(* CODESYS project SMB_Client_Visu.project

Project tree, tasks and I/O mapping:
  Device : CODESYS Control for Raspberry Pi, 3S - Smart Software Solutions GmbH, version 3.5.12.0
    application Application
      libraries: Standard, * (System); Standard64, * (System); BASIC, 3.3.3.0 (OSCAT); File Access, 3.5.7.0 (3S - Smart Software Solutions GmbH); VisuDialogs, * (System); Network, 3.5.7.0 (3S - Smart Software Solutions GmbH); Memory, 3.5.7.0 (3S - Smart Software Solutions GmbH)
      task MainTask (cyclic, interval 4 ms, priority 1) calls PLC_PRG
      task VISU_TASK (cyclic, interval 100 ms, priority 31) calls VisuElems.Visu_Prg
      visualisation Start
      visualisation SMB_Explorer
      Bausteine/
        program PLC_PRG [CFC]
        SMB2_Client/
          Explorer/
            data type Explorer
            data type Explorer_Dummy
          Misc/
            function block DER_Encoding [ST]
            function block DER_Len [ST]
            function WSTRING_UPPER [ST]
          NTLM/
            Struct/
              data type AUTHENTICATE_MESSAGE
              data type AVPairList
              data type CHALLENGE_MESSAGE
              data type NEGOTIATE_MESSAGE
              data type SessionData
            Functions/
              Hash/Encryption/
                function block HMAC_MD5 [ST]
                function block MD4 [ST]: ROUND1, ROUND2, ROUND3
                function block RC4 [ST]
              function block ComputeResponse [ST]
              function EncryptedSessionKey [ST]
              function block GenerateAuthenticateMessage [ST]
              function GetAVPairList [ST]
              function block LMOWFv2 [ST]
              function block mechListMIC [ST]
              function block MIC [ST]
              function block NTLM [ST]
              function block NTOWFv2 [ST]
              function block ProcessChallengeMessage [ST]
              function block SEALKEY [ST]
              function SetAVPairList [ST]
              function block SIGNKEY [ST]
          SMB2/
            Functions/
              function block ReadFile [ST]
              function block SendFile [ST]
              function NetShareEnumAll [ST]
              function NetShareBind [ST]
              function decodeSharePath [ST]
              Requests/
                function CloseReq [ST]
                function CreateReq [ST]
                function LogOffReq [ST]
                function QueryDirReq [ST]
                function TreeConnectReq [ST]
                function TreeDisconnectReq [ST]
                function ReadRequest [ST]
                function NegotiateReq [ST]
            Struct/
              data type Connection
              data type Open
              data type Session
              data type SMB_Client_Error
              SMB2_Requests/
                data type SMB_COM_NEGOTIATE
                data type SMB_Dialect
                data type SMB2_CLOSE_Request
                data type SMB2_CREATE_Request
                data type SMB2_LOGOFF_Request
                data type SMB2_QUERY_DIRECTORY_Request
                data type SMB2_READ_Request
                data type SMB2_SESSION_SETUP_Request
                data type SMB2_TREE_CONNECT_Request
                data type SMB2_TREE_DISCONNECT_Request
                data type SMB2_WRITE_Request
                data type SMB2_IOCTL_Request
              SMB2_Responses/
                data type SMB2_CLOSE_Response
                data type SMB2_CREATE_Reponse
                data type SMB2_LOGOFF_Response
                data type SMB2_NEGOTIATE_Response
                data type SMB2_READ_Response
                data type SMB2_SESSION_SETUP_Response
                data type SMB2_TREE_CONNECT_Response
                data type SMB2_TREE_DISCONNECT_Response
                data type SMB2_WRITE_Response
                data type SMB2_QUERY_DIRECTORY_Response
              data type TreeConnect
              data type SMB2_FileDirectoryInfo
              data type sharePath
              Header/
                data type SMB_Header
                data type SMB2_Header_Sync
                data type SMB2_Transport_Header
          global variables Constants
          function block SMB2_Client [ST]
          global variables VAR_Explorer
    SoftMotion General Axis Pool
    I²C
    SPI
    GPIOs_A_B : GPIOs A/B, 3S - Smart Software Solutions GmbH, version 3.5.11.0
        unmapped channels: digital inputs (GPIO0..GPIO31), digital outputs (GPIO0..GPIO31)
    Onewire
    Camera device
      <Leer>
  text list GlobalTextList
*)

// Device/Application/Bausteine/SMB2_Client/Explorer/Explorer
TYPE Explorer :
STRUCT
	xExecute:BOOL:=FALSE;
	IPAdress:STRING(80):='192.168.100.150';
	User:WSTRING(80):="UserName"; // UserName Default for Guest
	Password:WSTRING(80):=""; // Password Default for Guest
	UserDomain:WSTRING(80):="CoDeSys"; // Default 
	Login:BOOL; // WebVisu Button Login
	Logout:BOOL; // WebVisu Button Logout
	open:BOOL; // WebVisu Button open
	apply:BOOL; //Button übernehmen
	folderUp:BOOL; // WebVisu Button Folder Up
	openIndex:INT; // WebVisu Index of Directory
	applyIndex:INT;	// WebVisu Index for Apply Button
	write_read:INT:=1; // Write Read Direction
	write:BOOL:=TRUE; // WebVisu Indicator for Direction
	read:BOOL:=FALSE; // WebVisu Indicator for Direction
	sharePathDecoded:sharePath;
	DirectoryIndex:INT;
	folderDepth:INT; // Depth of shared Folder - 0 = NetshareNames, >0 = Directory Names
	online:BOOL:=TRUE; // WebVisu Online Indicator
	error:BOOL:=TRUE; // WebVisu Error Indicator
	busy:BOOL; // WebVisu Busy Indicator
	done:BOOL; // WebVisu Done Indicator
	start:bool; // WebVisu Start Transfer
	Directory:ARRAY[0..127] OF WSTRING(128); // List of Shares, Directory and Files
	xdir:ARRAY[0..127] OF BOOL; // Indicates Director (0 = Dir, 1= no dir)
	xfile:ARRAY[0..127] OF BOOL; // Indicates File (0 = File, 1= no File)
	actualsharePath:WSTRING(512); // 
	copysharePath:WSTRING(512); // Sharepath on PC for automatic mode
	plcPath:STRING(512):='/var/opt/codesys/datei.xyz'; // Path on PLC SD-Card
END_STRUCT
END_TYPE

// Device/Application/Bausteine/SMB2_Client/Explorer/Explorer_Dummy
// Dummy Struct for SMB2 Client without Explorer Mode all Arrays are short for memory saving

TYPE Explorer_Dummy :
STRUCT
	xExecute:BOOL:=FALSE;
	IPAdress:STRING(80):='192.168.100.150';
	User:WSTRING(80):="UserName"; // UserName Default for Guest
	Password:WSTRING(80):=""; // Password Default for Guest
	UserDomain:WSTRING(80):="CoDeSys"; // Default 
	Login:BOOL; // WebVisu Button Login
	Logout:BOOL; // WebVisu Button Logout
	open:BOOL; // WebVisu Button open
	apply:BOOL; //Button übernehmen
	folderUp:BOOL; // WebVisu Button Folder Up
	openIndex:INT; // WebVisu Index of Directory
	applyIndex:INT;	// WebVisu Index for Apply Button
	write_read:INT:=1; // Write Read Direction
	write:BOOL:=TRUE; // WebVisu Indicator for Direction
	read:BOOL:=FALSE; // WebVisu Indicator for Direction
	sharePathDecoded:sharePath;
	DirectoryIndex:INT;
	folderDepth:INT; // Depth of shared Folder - 0 = NetshareNames, >0 = Directory Names
	online:BOOL:=TRUE; // WebVisu Online Indicator
	error:BOOL:=TRUE; // WebVisu Error Indicator
	busy:BOOL; // WebVisu Busy Indicator
	done:BOOL; // WebVisu Done Indicator
	start:bool; // WebVisu Start Transfer
	Directory:ARRAY[0..1] OF WSTRING(1); // List of Shares, Directory and Files
	xdir:ARRAY[0..1] OF BOOL; // Indicates Director (0 = Dir, 1= no dir)
	xfile:ARRAY[0..1] OF BOOL; // Indicates File (0 = File, 1= no File)
	actualsharePath:WSTRING(1); // 
	copysharePath:WSTRING(1); // Sharepath on PC for automatic mode
	plcPath:STRING(1); // Path on PLC SD-Card

END_STRUCT
END_TYPE

// Device/Application/Bausteine/SMB2_Client/NTLM/Struct/AUTHENTICATE_MESSAGE
{attribute 'pack_mode' := '1'} (*aligned to byte*)

TYPE AUTHENTICATE_MESSAGE :
STRUCT
	Signature:STRING(7):='NTLMSSP';
	MessageType:DWORD:=16#0003;
	// LmChallengeResponse
	LmChallengeResponseLen:WORD;
	LmChallengeResponseMaxLen:WORD;
	LmChallengeResponseBufferOffset:DWORD;
	// NtChallengeResponse
	NtChallengeResponseLen:WORD;
	NtChallengeResponseMaxLen:WORD;
	NtChallengeResponseBufferOffset:DWORD;
	// Domain Name
	DomainNameLen:WORD;
	DomainNameMaxLen:WORD;
	DomainNameBufferOffset:DWORD;
	// User Name
	UserNameLen:WORD;
	UserNameMaxLen:WORD;
	UserNameBufferOffset:DWORD;
	// Workstation
	WorkstationLen:WORD;
	WorkstationMaxLen:WORD;
	WorkstationBufferOffset:DWORD;
	// EncryptedRandomSessionKey
	EncryptedRandomSessionKeyLen:WORD;
	EncryptedRandomSessionKeyMaxLen:WORD;
	EncryptedRandomSessionKeyBufferOffset:DWORD;
	//
	NegotiateFlags:DWORD; // Negotiate Flags
	Version:ARRAY[0..1] OF DWORD:=[16#3839000A, 16#F0000000]; // Verson Number
	MIC:ARRAY[0..15] OF BYTE; // Message Integrity Code
	Payload:ARRAY[0..1023] OF BYTE; // Payload for Names and Attributes
	PayLoadSize:INT; // Length of Payload
END_STRUCT
END_TYPE

// Device/Application/Bausteine/SMB2_Client/NTLM/Struct/AVPairList
TYPE AVPairList :
STRUCT
	NBComputerName:WSTRING(80); // 
	NBDomainName:WSTRING(80);
	DNSComputerName:WSTRING(80);
	DNSDomainName:WSTRING(80);
	xTimeStamp:BOOL; // Timestamp is there
	TimeStamp:ARRAY[0..7] OF BYTE;
END_STRUCT
END_TYPE

// Device/Application/Bausteine/SMB2_Client/NTLM/Struct/CHALLENGE_MESSAGE
{attribute 'pack_mode' := '1'} (*aligned to byte*)

TYPE CHALLENGE_MESSAGE :
STRUCT
	Signature:STRING(7); // NTLMSSP
	MessageType:DWORD; // Challenge MEssage
	// TargetNameFields
	TargetNameLen:WORD;
	TargetNameMaxLen:WORD;
	TargetNameBufferOffset:DWORD;
	//
	NegotiateFlags:DWORD; // NEgotiate Flags
	ServerChallenge:ARRAY[0..7] OF BYTE; // Random Numbers Server Challenge
	Reserved:ARRAY[0..7] OF BYTE;
	// TargetInfoFields
	TargetInfoLen:WORD;
	TargetInfoMaxLen:WORD;
	TargetInfoBufferOffset:DWORD;
	//
	Version:ARRAY[0..1] OF DWORD; // Version Number
	// Payload
	TargetName:WSTRING(80);
	AVPairList:AVPairList;
	AVPairListPayload:ARRAY[0..255] OF BYTE;
END_STRUCT
END_TYPE

// Device/Application/Bausteine/SMB2_Client/NTLM/Struct/NEGOTIATE_MESSAGE
{attribute 'pack_mode' := '1'} (*aligned to byte*)

TYPE NEGOTIATE_MESSAGE :
STRUCT
	Signature:STRING(7):= 'NTLMSSP'; // NTLMSSP
	MessageType:DWORD:=16#00000001; // Negotiate MEssage
	NegotiateFlags:DWORD; // Negotiate Flags
	// Doman Name
	DomainNameLen:WORD; 
	DomainNameMaxLen:WORD;
	DomainNameBufferOffset:DWORD;
	// Workstation Name
	WorkstationLen:WORD;
	WorkstationMaxLen:WORD;
	WorkstationBufferOffset:DWORD;
	Version:ARRAY[0..1] OF DWORD:=[16#3839000a, 16#F0000000] ; // Version
END_STRUCT
END_TYPE

// Device/Application/Bausteine/SMB2_Client/NTLM/Struct/SessionData
TYPE SessionData :
STRUCT
//	mode Mode

	user:WSTRING(80); // Username
	password:WSTRING(80); // Password
	userDomain:WSTRING(80); // User Doman

	NegotiateFlags:DWORD; // Negotiate Flags

	negotiateMessage:POINTER TO NEGOTIATE_MESSAGE; // Pointer to Negotiate Message
	challengeMessage:POINTER TO CHALLENGE_MESSAGE; // Pointer to Challenge Message
//	authenticateMessage *AuthenticateMessage

	serverChallenge:ARRAY[0..7] OF BYTE; // Server Challenge random number
	clientChallenge:ARRAY[0..7] OF BYTE; // client Challenge for response
	ntChallengeResponse:ARRAY[0..511] OF BYTE; // NT Challenge Response
	ntChallengeResponseLen:WORD;  // Length of NT Challenge Response
	lmChallengeResponse:ARRAY[0..511] OF BYTE;  // LM Challenge Response
	lmChallengeResponseLen:WORD; // Length of LM Challenge Response

	responseKeyLM: ARRAY[0..15] OF BYTE; // Response Key LM for calculation
	responseKeyNT: ARRAY[0..15] OF BYTE; // Response Key NT for calculation
	exportedSessionKey: ARRAY[0..15] OF BYTE; // exported Session Key
	encryptedRandomSessionKey: ARRAY[0..15] OF BYTE; // encrypted Random Session Key
	keyExchangeKey:ARRAY[0..15] OF BYTE; // Key Exchange Key
	sessionBaseKey:ARRAY[0..15] OF BYTE; // Session Base Key
	mic                 :ARRAY[0..15] OF BYTE; // Message Integrity Code

	ClientSigningKey: ARRAY[0..15] OF BYTE; // Client Signing Key
	ServerSigningKey: ARRAY[0..15] OF BYTE; // Server Signing Key
	ClientSealingKey: ARRAY[0..15] OF BYTE; // Client Sealing Key
	ServerSealingKey: ARRAY[0..15] OF BYTE; // Server Sealing Key

	clientHandle:RC4;
	serverHandle:RC4;
	
	NegMessByte:ARRAY[0..511] OF BYTE;
	NegMessByteLen:INT;
	ChallMessByte:ARRAY[0..511] OF BYTE;
	ChallMessByteLen:INT;
	AuthMessByte:ARRAY[0..511] OF BYTE;
	AuthMessByteLen:INT;
	
	mechListMIC:ARRAY[0..19] OF BYTE;
END_STRUCT
END_TYPE

// Device/Application/Bausteine/SMB2_Client/SMB2/Struct/Connection
TYPE Connection :
STRUCT
	Session:Session; // Parameter of active Session
	MaxTransactSize:DWORD; // Max Transaction Size
	MaxReadSize:DWORD; // Max Read Size from Server
	MaxWriteSize:DWORD;	// Max Write Size to Server
	MessageID: ARRAY[0..1] OF DWORD; // Sequence Number
	ServerGuid:ARRAY [0..3] OF DWORD; // Server global unique identifier
	RequireSigning:BOOL;
	LastStatus:DWORD; // Last Status of Response
	ServerName:STRING(80); // Servername
	wServerName:WSTRING(80); // Servername Unicode String
	User:WSTRING(80); // Username
	Password:WSTRING(80); // Password
	UserDomain:WSTRING(80); // User Domain
	requestedFileName:WSTRING(512); // requested File Name
END_STRUCT
END_TYPE

// Device/Application/Bausteine/SMB2_Client/SMB2/Struct/Open
TYPE Open :
STRUCT
	FileId:ARRAY[0..3] OF DWORD; // File ID of opened File (After Create Request)
	FileSize:ARRAY[0..1] OF DWORD; // File Size of opened File (After Create Request)
	ReadDataOffset:BYTE; // Actual Offset in opened File
	ReadDataLength:DWORD; // Actual Size of read Data
END_STRUCT
END_TYPE

// Device/Application/Bausteine/SMB2_Client/SMB2/Struct/Session
TYPE Session :
STRUCT
	SessionID:ARRAY[0..1] OF DWORD; // Session ID of active Session
	TreeConnect: TreeConnect; // Parameter of Active Tree
	SessionKey:ARRAY[0..15] OF BYTE; 
	SigningRequired:BOOL;
	Open:Open;
END_STRUCT
END_TYPE

// Device/Application/Bausteine/SMB2_Client/SMB2/Struct/SMB_Client_Error
TYPE SMB_Client_Error :
STRUCT
	Error_1:INT; // Error Step in SMB2 Client 
	Error_2:DWORD; // Error/Status from Response
	TCP:NBS.ERROR; // Error TCP Function
	ConRST:BOOL; // Connection Reset from Server
END_STRUCT
END_TYPE

// Device/Application/Bausteine/SMB2_Client/SMB2/Struct/SMB2_Requests/SMB_COM_NEGOTIATE
{attribute 'pack_mode' := '1'} (*aligned to byte*)

TYPE SMB_COM_NEGOTIATE :	
STRUCT
	WORDCOUNT :BYTE;
	BYTECOUNT :WORD;
	Dialects: ARRAY[0..8] OF SMB_Dialect;
END_STRUCT
END_TYPE

// Device/Application/Bausteine/SMB2_Client/SMB2/Struct/SMB2_Requests/SMB_Dialect
{attribute 'pack_mode' := '1'} (*aligned to byte*)

TYPE SMB_Dialect :
STRUCT
	BufferFormat:BYTE;
	DialectString:STRING;
END_STRUCT
END_TYPE

// Device/Application/Bausteine/SMB2_Client/SMB2/Struct/Header/SMB_Header
{attribute 'pack_mode' := '1'} (*aligned to byte*)

TYPE SMB_Header :
STRUCT
	Protocol: ARRAY[0..3] OF BYTE;
	Command: BYTE;
	Status:DWORD;
	Flags:BYTE;
	Flags2:WORD;
	PIDHigh:WORD;
	SecurityFeatures:ARRAY[0..7] OF BYTE;
	Reserved:WORD;
	TID:WORD;
	PIDLow:WORD;
	UID:WORD;
	MID:WORD;
END_STRUCT
END_TYPE

// Device/Application/Bausteine/SMB2_Client/SMB2/Struct/Header/SMB2_Header_Sync
// [MS-SMB2] 2.2.1.2
{attribute 'pack_mode' := '1'} (*aligned to byte*)

TYPE SMB2_Header_Sync :
STRUCT
	ProtocolID: ARRAY[0..3] OF BYTE;
	StructureSize:WORD:=64;
	CreditCharge:WORD;
	Status:DWORD;
	Command:WORD;
	CreditRepReq:WORD;
	Flags: DWORD;
	NextCommand:DWORD;
	MessageID: ARRAY[0..1] OF DWORD;
	Reserved: DWORD;
	TreeID:DWORD;
	SessionID: ARRAY[0..1] OF DWORD;
	Signature: ARRAY[0..3] OF DWORD;
END_STRUCT
END_TYPE

// Device/Application/Bausteine/SMB2_Client/SMB2/Struct/SMB2_Requests/SMB2_CLOSE_Request
// [MS-SMB2] 2.2.15

{attribute 'pack_mode' := '1'} (*aligned to byte*)

TYPE SMB2_CLOSE_Request :
STRUCT
	StructureSize:WORD:=24;
	Flags:WORD;
	Reserved:DWORD:=0;
	FileId:ARRAY[0..3] OF DWORD;
END_STRUCT
END_TYPE

// Device/Application/Bausteine/SMB2_Client/SMB2/Struct/SMB2_Requests/SMB2_CREATE_Request
// [MS-SMB2] 2.2.13

{attribute 'pack_mode' := '1'} (*aligned to byte*)

TYPE SMB2_CREATE_Request :
STRUCT
	StructureSize:WORD:=57;
	SecurityFlags:BYTE;
	RequestedOplockLevel:BYTE;
	ImpersonationLevel:DWORD;
	SmbCreateFlags:ARRAY[0..1] OF DWORD;
	Reserved:ARRAY[0..1] OF DWORD;
	DesiredAccess:DWORD;
	FileAttributes:DWORD;
	ShareAccess:DWORD;
	CreateDisposition:DWORD;
	CreateOptions:DWORD;
	NameOffset:WORD;
	NameLength:WORD;
	CreateContextsOffset:DWORD;
	CreateContextsLength:DWORD;
	Payload:ARRAY[0..255] OF BYTE;
END_STRUCT
END_TYPE

// Device/Application/Bausteine/SMB2_Client/SMB2/Struct/SMB2_Requests/SMB2_LOGOFF_Request
// [MS-SMB2] 2.2.7

{attribute 'pack_mode' := '1'} (*aligned to byte*)

TYPE SMB2_LOGOFF_Request :
STRUCT
	StructureSize:WORD;
	Reserved:WORD;
END_STRUCT
END_TYPE

// Device/Application/Bausteine/SMB2_Client/SMB2/Struct/SMB2_Requests/SMB2_QUERY_DIRECTORY_Request
// [MS-SMB2] 2.2.33

{attribute 'pack_mode' := '1'} (*aligned to byte*)

TYPE SMB2_QUERY_DIRECTORY_Request :
STRUCT
	StructureSize:WORD:=33;
	FileInformationClass:BYTE;
	Flags:BYTE;
	FileIndex:DWORD;
	FileId:ARRAY[0..3] OF DWORD;
	FileNameOffset:WORD;
	FileNameLength:WORD;
	OutputbufferLength:DWORD;
	Payload:ARRAY[0..127] OF BYTE;
END_STRUCT
END_TYPE

// Device/Application/Bausteine/SMB2_Client/SMB2/Struct/SMB2_Requests/SMB2_READ_Request
// [MS-SMB2] 2.2.19

{attribute 'pack_mode' := '1'} (*aligned to byte*)

TYPE SMB2_READ_Request :
STRUCT
	StructureSize:WORD:=49;
	Padding:BYTE; // Offset in Response from Header Start ( for data optimization)
	Flags:BYTE:=0; // Not used in SMB 2
	Length:DWORD; // Length of data to read
	Offset:LWORD; // Offset in File
	FileId:ARRAY[0..3] OF DWORD;
	MinimumCount:DWORD; // Minimal number of Bytes to be read for success
	Channel:DWORD:=0; // SMB2 = 0;
	RemainingBytes:DWORD; // Number of Bytes to be read after this operation completes
	ReadChannelInfoOffset:WORD:=0; // SMB2 = 0;
	ReadChannelInfoLength:WORD:=0; // SMB2 = 0;
END_STRUCT
END_TYPE

// Device/Application/Bausteine/SMB2_Client/SMB2/Struct/SMB2_Requests/SMB2_SESSION_SETUP_Request
// [MS-SMB2] 2.2.5

{attribute 'pack_mode' := '1'} (*aligned to byte*)

TYPE SMB2_SESSION_SETUP_Request :
STRUCT
	StructureSize:WORD;
	Flags:BYTE;
	SecurityMode:BYTE;
	Capabilities:DWORD;
	Channel:DWORD;
	SecurityBufferOffset:WORD;
	SecurityBufferLength:WORD;
	PrevSessionsId:ARRAY[0..1] OF DWORD;
END_STRUCT
END_TYPE

// Device/Application/Bausteine/SMB2_Client/SMB2/Struct/SMB2_Requests/SMB2_TREE_CONNECT_Request
// [MS-SMB2] 2.2.9

{attribute 'pack_mode' := '1'} (*aligned to byte*)

TYPE SMB2_TREE_CONNECT_Request :
STRUCT
	StructureSize:WORD;
	Flags:WORD;
	PathOffset:WORD;
	PathLength:WORD;
	PathName:WSTRING(256);
END_STRUCT
END_TYPE

// Device/Application/Bausteine/SMB2_Client/SMB2/Struct/SMB2_Requests/SMB2_TREE_DISCONNECT_Request
// [MS-SMB2] 2.2.11

{attribute 'pack_mode' := '1'} (*aligned to byte*)

TYPE SMB2_TREE_DISCONNECT_Request :
STRUCT
	StructureSize:WORD;
	Reserved:WORD;
END_STRUCT
END_TYPE

// Device/Application/Bausteine/SMB2_Client/SMB2/Struct/SMB2_Requests/SMB2_WRITE_Request
// [MS-SMB2] 2.2.21

{attribute 'pack_mode' := '1'} (*aligned to byte*)

TYPE SMB2_WRITE_Request :
STRUCT
	StructureSize:WORD:=49;
	DataOffset:WORD;
	Length:DWORD;
	Offset:LWORD;
	FileId:ARRAY[0..3] OF DWORD;
	Channel:DWORD:=0; // SMB2 = 0;
	RemainingBytes:DWORD;
	WriteChannelInfoOffset:WORD:=0; // SMB2 = 0;
	WriteChannelInfoLength:WORD:=0; // SMB2 = 0;
	Flags:DWORD:=0; // SMB2 = 0;
END_STRUCT
END_TYPE

// Device/Application/Bausteine/SMB2_Client/SMB2/Struct/SMB2_Responses/SMB2_CLOSE_Response
// [MS-SMB2] 2.2.16

{attribute 'pack_mode' := '1'} (*aligned to byte*)

TYPE SMB2_CLOSE_Response :
STRUCT
	StructureSize:WORD;
	Flags:WORD;
	Reserved:DWORD;
	CreateionTime:ARRAY[0..1] OF DWORD;
	LastAccessTime:ARRAY[0..1] OF DWORD;
	LastWriteTime:ARRAY[0..1] OF DWORD;
	ChangeTime:ARRAY[0..1] OF DWORD;
	AllocationSize:ARRAY[0..1] OF DWORD;
	EndofFile:ARRAY[0..1] OF DWORD;
	FileAttributes:DWORD;
END_STRUCT
END_TYPE

// Device/Application/Bausteine/SMB2_Client/SMB2/Struct/SMB2_Responses/SMB2_CREATE_Reponse
// [MS-SMB2] 2.2.114

{attribute 'pack_mode' := '1'} (*aligned to byte*)

TYPE SMB2_CREATE_Reponse :
STRUCT
	StructureSize:WORD;
	OplockLevel:BYTE;
	Flags:BYTE;
	CreateAction:DWORD;
	CreateionTime:ARRAY[0..1] OF DWORD;
	LastAccessTime:ARRAY[0..1] OF DWORD;
	LastWriteTime:ARRAY[0..1] OF DWORD;
	ChangeTime:ARRAY[0..1] OF DWORD;
	AllocationSize:ARRAY[0..1] OF DWORD;
	EndofFile:ARRAY[0..1] OF DWORD;
	FileAttributes:DWORD;
	Reserved2:DWORD;
	FileId:ARRAY[0..3] OF DWORD;
	CreateContextsOffset:DWORD;
	CreateContextsLength:DWORD;
END_STRUCT
END_TYPE

// Device/Application/Bausteine/SMB2_Client/SMB2/Struct/SMB2_Responses/SMB2_LOGOFF_Response
// [MS-SMB2] 2.2.8

{attribute 'pack_mode' := '1'} (*aligned to byte*)

TYPE SMB2_LOGOFF_Response :
STRUCT
	StructureSize:WORD;
	Reserved:WORD;
END_STRUCT
END_TYPE

// Device/Application/Bausteine/SMB2_Client/SMB2/Struct/SMB2_Responses/SMB2_NEGOTIATE_Response
// [MS-SMB2] 2.2.4

{attribute 'pack_mode' := '1'} (*aligned to byte*)

TYPE SMB2_NEGOTIATE_Response :
STRUCT
	StructureSize:WORD;
	SecurityMode:WORD;
	DialectRevision:WORD;
	NegotiateContextCount:WORD;
	ServerGuid:ARRAY [0..3] OF DWORD;
	Capabilities:DWORD;
	MaxTransactSize:DWORD;
	MaxReadSize:DWORD;
	MaxWriteSize:DWORD;
	SystemTime:ARRAY[0..1] OF DWORD;
	ServerStartTime:ARRAY[0..1] OF DWORD;
	SecurityBufferOffset:WORD;
	SecurityBufferLength:WORD;
	NegotiateContextOffset:DWORD;
	
END_STRUCT
END_TYPE

// Device/Application/Bausteine/SMB2_Client/SMB2/Struct/SMB2_Responses/SMB2_READ_Response
// [MS-SMB2] 2.2.20

{attribute 'pack_mode' := '1'} (*aligned to byte*)

TYPE SMB2_READ_Response :
STRUCT
	StructureSize:WORD;
	DataOffset:BYTE; // Data Offset in Response Buffer from SMB2 Header
	Reserved:BYTE;
	DataLength:DWORD;
	DataRemaining:DWORD;
	Reserved2:DWORD;
END_STRUCT
END_TYPE

// Device/Application/Bausteine/SMB2_Client/SMB2/Struct/SMB2_Responses/SMB2_SESSION_SETUP_Response
// [MS-SMB2] 2.2.6

{attribute 'pack_mode' := '1'} (*aligned to byte*)

TYPE SMB2_SESSION_SETUP_Response :
STRUCT
	StructureSize:WORD;
	SessionFlags:WORD;
	SecurityBufferOffset:WORD;
	SecurityBufferLength:WORD;
END_STRUCT
END_TYPE

// Device/Application/Bausteine/SMB2_Client/SMB2/Struct/SMB2_Responses/SMB2_TREE_CONNECT_Response
// [MS-SMB2] 2.2.10

{attribute 'pack_mode' := '1'} (*aligned to byte*)

TYPE SMB2_TREE_CONNECT_Response :
STRUCT
	StructureSize:WORD;
	ShareType:BYTE;
	Reserved:BYTE;
	ShareFlags:DWORD;
	Capabilities:DWORD;
	MaxmalAccess:DWORD;
END_STRUCT
END_TYPE

// Device/Application/Bausteine/SMB2_Client/SMB2/Struct/SMB2_Responses/SMB2_TREE_DISCONNECT_Response
// [MS-SMB2] 2.2.12

{attribute 'pack_mode' := '1'} (*aligned to byte*)

TYPE SMB2_TREE_DISCONNECT_Response :
STRUCT
	StructureSize:WORD;
	Reserved:WORD;
END_STRUCT
END_TYPE

// Device/Application/Bausteine/SMB2_Client/SMB2/Struct/SMB2_Responses/SMB2_WRITE_Response
// [MS-SMB2] 2.2.22

{attribute 'pack_mode' := '1'} (*aligned to byte*)

TYPE SMB2_WRITE_Response :
STRUCT
	StructureSize:WORD;
	Reserved:WORD; 
	Count:DWORD; // Number of written Bytes
	Remaining:DWORD; // Must be 0
	WriteChannelInfoOffset:WORD; // Must be 0
	WriteChannelInfoLength:WORD; // Must be 0
END_STRUCT
END_TYPE

// Device/Application/Bausteine/SMB2_Client/SMB2/Struct/Header/SMB2_Transport_Header
// [MS-SMB2] 2.1

{attribute 'pack_mode' := '1'} (*aligned to byte*)

TYPE SMB2_Transport_Header :
STRUCT
	Zero:BYTE; (*Always Zero, for Direct TCP Transport*)
	StreamProtocolLength:UDINT; (*Length of SMB2 Packet without Transport Header*)
END_STRUCT
END_TYPE

// Device/Application/Bausteine/SMB2_Client/SMB2/Struct/TreeConnect
TYPE TreeConnect :
STRUCT
	ShareName:WSTRING(128); // Name of Share Name
	TreeConnectId:DWORD; // TreeID of opened Tree
	IsDfsShare:BOOL;
END_STRUCT
END_TYPE

// Device/Application/Bausteine/SMB2_Client/SMB2/Struct/SMB2_FileDirectoryInfo
{attribute 'pack_mode' := '1'} (*aligned to byte*)

TYPE SMB2_FileDirectoryInfo :
STRUCT
	NextOffset:DWORD; // Offset to Next File Directory Info
	FileIndex:DWORD; // File Index Number
	Create:LWORD; // Create Time
	LastAcc:LWORD; // Last Access Time
	LastWrite:LWORD; // Last Write Time
	LastChange:LWORD; // Last Change Time
	EndOfFile:LWORD; // End of File in Byte
	AllocSize:LWORD; // Allocation Size on Disk
	FileAtr:DWORD; // File Attributes
	FileNameLength:DWORD; // Length of File Name
END_STRUCT
END_TYPE

// Device/Application/Bausteine/SMB2_Client/SMB2/Struct/SMB2_Responses/SMB2_QUERY_DIRECTORY_Response
// [MS-SMB2] 2.2.34

{attribute 'pack_mode' := '1'} (*aligned to byte*)

TYPE SMB2_QUERY_DIRECTORY_Response :
STRUCT
	StructureSize:WORD;
	OutputBufferOffset:WORD;
	OutputBufferLength:DWORD;
END_STRUCT
END_TYPE

// Device/Application/Bausteine/SMB2_Client/SMB2/Struct/SMB2_Requests/SMB2_IOCTL_Request
// [MS-SMB2] 2.2.31

{attribute 'pack_mode' := '1'} (*aligned to byte*)

TYPE SMB2_IOCTL_Request :
STRUCT
	StructureSize:WORD;
	Reserved:WORD;
	CtlCode:DWORD;
	FileID:ARRAY[0..3] OF DWORD;
	InputOffset:DWORD;
	InputCount:DWORD;
	MaxInputResponse:DWORD;
	OutputOffset:DWORD;
	OutputCount:DWORD;
	MaxOutputResponse:DWORD;
	Flags:DWORD;
	Reserved2:DWORD;
END_STRUCT
END_TYPE

// Device/Application/Bausteine/SMB2_Client/SMB2/Struct/sharePath
TYPE sharePath :
STRUCT
	serverName:WSTRING(64); // ServerName or IP Adress - max 64 Symbols
	treeName:WSTRING(256); // ShareName of shared Folder - max 256 Symbols
	fileName:WSTRING(512); // Filename - \folder\folder_2\filename.x
END_STRUCT
END_TYPE

// Device/Application/Bausteine/SMB2_Client/Constants
{attribute 'qualified_only'}
VAR_GLOBAL CONSTANT
	(*SMB2 Header Commands*)
	NEGOTIATE 			:UINT:= 16#0000;
	SESSION_SETUP 		:UINT:= 16#0001;
	LOGOFF 				:UINT:= 16#0002;
	TREE_CONNECT 		:UINT:= 16#0003;
	TREE_DISCONNECT 	:UINT:= 16#0004;
	CREATE 				:UINT:= 16#0005;
	CLOSE 				:UINT:= 16#0006;
	FLUSH 				:UINT:= 16#0007;
	READ 				:UINT:= 16#0008;
	WRITE 				:UINT:= 16#0009;
	LOCK 				:UINT:= 16#000A;
	IOCTL 				:UINT:= 16#000B;
	CANCEL 				:UINT:= 16#000C;
	ECHO 				:UINT:= 16#000D;
	QUERY_DIRECTORY 	:UINT:= 16#000E;
	CHANGE_NOTIFY 		:UINT:= 16#000F;
	QUERY_INFO 			:UINT:= 16#0010;
	SET_INFO 			:UINT:= 16#0011;
	OPLOCK_BREAK 		:UINT:= 16#0012;
	(*SMB2 Header Flags*)
	SMB2_FLAGS_SERVER_TO_REDIR 			:UDINT:= 16#00000001;
	SMB2_FLAGS_ASYNC_COMMAND 			:UDINT:= 16#00000002;
	SMB2_FLAGS_RELATED_OPERATIONS 		:UDINT:= 16#00000004;
	SMB2_FLAGS_SIGNED 					:UDINT:= 16#00000008;
	SMB2_FLAGS_PRIORITY_MASK 			:UDINT:= 16#00000070;
	SMB2_FLAGS_DFS_OPERATIONS 			:UDINT:= 16#10000000;
	SMB2_FLAGS_REPLAY_OPERATION 		:UDINT:= 16#20000000;
	
	(*SMB Flags*)
	SMB_FLAGS_LOCK_AND_READ_OK 			:USINT:= 16#01;
	SMB_FLAGS_BUF_AVAIL 				:USINT:= 16#02;
	SMB_FLAGS_CASE_INSENSITIVE 			:USINT:= 16#08;
	SMB_FLAGS_CANONICALIZED_PATHS 		:USINT:= 16#10;
	SMB_FLAGS_OPLOCK 					:USINT:= 16#20;
	SMB_FLAGS_OPBATCH 					:USINT:= 16#40;
	SMB_FLAGS_REPLY						:USINT:= 16#80;
	
	SMB_FLAGS2_LONG_NAMES				:UINT:= 16#0001;
	SMB_FLAGS2_EAS						:UINT:= 16#0002;
	SMB_FLAGS2_SMB_SECURITY_SIGNATURE 	:UINT:= 16#0004;
	SMB_FLAGS2_IS_LONG_NAME				:UINT:= 16#0040;
	SMB_FLAGS2_DFS						:UINT:= 16#1000;
	SMB_FLAGS2_PAGING_IO 				:UINT:= 16#2000;
	SMB_FLAGS2_NT_STATUS 				:UINT:= 16#4000;
	SMB_FLAGS2_UNICODE 					:UINT:= 16#8000;
	
	(*Header Status*)
	STATUS_SUCCESS						:UDINT:= 16#00000000;
	STATUS_MORE_PROCESSING_REQUIRED		:UDINT:= 16#C0000016;
END_VAR

// Device/Application/Bausteine/SMB2_Client/VAR_Explorer
{attribute 'qualified_only'}
VAR_GLOBAL RETAIN
	Visu_Explorer:explorer;
END_VAR

// Device/Application/Bausteine/PLC_PRG
PROGRAM PLC_PRG
VAR
	SMB2: SMB2_Client; // SMB2 Client
	start:BOOL; // Start for Automatic Mode (or for testing)
	done:BOOL;	// File Transfer Done or Explorer Mode LogOff Done
	busy:BOOL; // File Transfer active or Explorer Mode connected to Server
	error:BOOL; // Error
	eError:SMB_Client_Error; // Error Struct for detailed error information
END_VAR

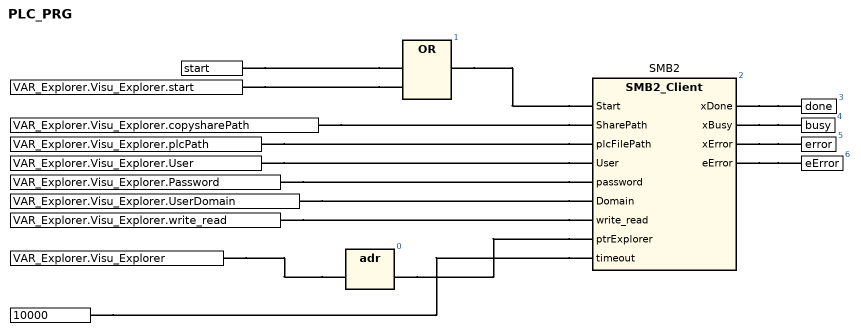
SMB2(
    Start := start OR VAR_Explorer.Visu_Explorer.start,
    SharePath := VAR_Explorer.Visu_Explorer.copysharePath,
    plcFilePath := VAR_Explorer.Visu_Explorer.plcPath,
    User := VAR_Explorer.Visu_Explorer.User,
    password := VAR_Explorer.Visu_Explorer.Password,
    Domain := VAR_Explorer.Visu_Explorer.UserDomain,
    write_read := VAR_Explorer.Visu_Explorer.write_read,
    ptrExplorer := adr(VAR_Explorer.Visu_Explorer),
    timeout := 10000); // SMB2_Client
done := SMB2.xDone;
busy := SMB2.xBusy;
error := SMB2.xError;
eError := SMB2.eError;

END_PROGRAM

// Device/Application/Bausteine/SMB2_Client/SMB2_Client
FUNCTION_BLOCK SMB2_Client
VAR_INPUT
	Start:BOOL;					// Starts Connection and Write/Read process
	SharePath:WSTRING(256);		// shared folder Path, with Ip Adress - \\IP Adress\share\subfolder\filename.x
	plcFilePath:STRING(256);	// Path and Name of File in the PLC - manufactur / OS specific
	User:WSTRING(80);			// User Name - for Guest choose any User Name
	password:WSTRING(80);		// User Password for User Name - "Password01" - for Guest use empty WSTRING ""
	Domain:WSTRING(80); 		// Domain Name of PLC, for default use "CoDeSys"
	write_read:INT; 			// 1 = write file from PLC Memory to Shared Folder , 2 = read file from Shared Folder to PLC Memory
	ptrExplorer:POINTER TO Explorer; // Pointer to Explorer Variable for WebVisu Explorer
	timeout:UINT; // Timeout in ms
END_VAR
VAR_OUTPUT
	xDone:BOOL; // send/receive done or explorer mode log off done
	xBusy:BOOL;	// send/receive busy or explorer mode active
	xError:BOOL; // error
	eError:SMB_Client_Error; // error struct for detailed error information
	
END_VAR
VAR
	ConnectionParam:Connection; // Connection Parameter
	sharePathDecoded:sharePath; // SharePath decoded in ServerName, TreeName and FileName
	explorerDummy:Explorer_Dummy; // Explorer Dummy Variable when no Explorer used
	explorerMode:BOOL; // Indicates Explorer active
	explorerVar:BOOL:=FALSE;
	
	step:INT;	// actual step
	lastStep:INT; // step last cycle - for timeout
	errorStep:INT; // step of error
	timeoutTON:TON; // timeout timer
	autoLogOffTON:TON; // Automactic LogOff in WebVisu after x Minutes
	
	lastActive:BOOL; // 
	(*Connection*)
	TCP1: NBS.TCP_Client; // TCP Client Funtcion
	hCon:CAA.handle; // Handle to TCP Connection, for read and write
	Erro: NBS.ERROR; // TCP Error
	active:BOOL; // Indicates active TCP connection
	(*Receive TCP*)
	TCPRECV: NBS.TCP_Read; // TCP Receive Function
	recvP:CAA.PVOID:=ADR(recvBuf); // Pointer to Receive Buffer
	recvBuf: ARRAY[0..BufferSize+1024] OF BYTE; // receive buffer
	recvComplete:BOOL; // Received and copied to Response Variables
	recvOK:BOOL; // All TCP Segments received, ready for copy to variables
	(*Receive fragmeted TCP Packets*)
	MessageLength:UDINT; // Message Length in Header
	recvLength:UDINT; // Received Data Length
	newBufferIndex:UDINT; // Start for next received data, used for fragmented TCP
	
	(*Write TCP*)
	TCPSEND: NBS.TCP_WRITE; // TCP Send Function
	sendBuf: ARRAY[0..BufferSize+1024] OF BYTE; // send buffer
	sendP: CAA.PVOID:=ADR(sendBuf); // Pointer to Send Buffer
	sendSize: CAA.SIZE; // Length of Send Buffer
	sendS:uint;
	startSend: BOOL; // Start Sending
	
	(*SMB Responses*)
	TransportHeader:SMB2_Transport_Header;
	TransportHeaderRep:SMB2_Transport_Header;
	SMB2Header: SMB2_Header_Sync;
	SMB2HeaderRep: SMB2_Header_Sync;
	SMBHeader: SMB_Header;
	SMBNegotiate:SMB_COM_NEGOTIATE;
	SMB2NegotiateRep:SMB2_NEGOTIATE_Response;
	SMB2SessionSetup:SMB2_SESSION_SETUP_Request;
	SMB2SessionSetupRep:SMB2_SESSION_SETUP_Response;
	SMB2TreeConnectRep:SMB2_TREE_CONNECT_Response;
	SMB2CreateRep:SMB2_CREATE_Reponse;
	SMB2ReadRep:SMB2_READ_Response;
	SMB2WriteRep:SMB2_WRITE_Response;
	SMB2CloseRep:SMB2_CLOSE_Response;
	SMB2DisconnectRep:SMB2_TREE_DISCONNECT_Response;
	SMB2LogoffRep:SMB2_LOGOFF_Response;
	SMB2QueryDirRep:SMB2_QUERY_DIRECTORY_Response;
	tmpFileDirectoryInfo:SMB2_FileDirectoryInfo;
	
	repSize:UINT; // Size of received Data - Transport Header
	repP:POINTER TO BYTE;
	tmpIndex:UINT;
	repIndex:UINT;
	startIndex:UINT;

	sendF:sendFile; // Send File to Server
	readF:ReadFile; // Receive File from Server
	NTLM:NTLM; // NTLM Function Block
	
	i:DINT;
	j:INT;
	h:INT;
	
	// explorer mode variable
	varPtr:POINTER TO ARRAY[0..9216] OF BYTE;
	stringPtr:POINTER TO ARRAY[0..1024] OF BYTE;
	tempOffset:DINT;	
	tempLen:UINT;
	numberOfNames:INT;	
	pVar:POINTER TO ARRAY[0..1024] OF BYTE;
	pWord:POINTER TO ARRAY[0..1024] OF WORD;
	pLWORD:POINTER TO ARRAY[0..7] OF BYTE;
	tempLWORD:LWORD;
	tempLWORD2:LWORD;
	tempwString:WSTRING(512);
END_VAR
VAR CONSTANT
	BufferSize:UDINT:= 16384;//8192//32768//16384 - Buffersize for send and receive Buffer
END_VAR

// This is the Main SMB2_Client Function
// Normal Mode: File Transfer in Both Direction PLC - > PC and PC -> PLC. Both diretions initiates by PLC.
// Explorer Mode in HMI for browsing trough Shared Folders and setting new Share Path for Automatic Mode.

// Timeout
timeoutTON(PT:=UINT_TO_TIME(timeout));

IF (step = laststep) AND NOT (step=01) AND NOT (step=500) THEN // Start Timer when same step
	timeoutTON.IN := TRUE;
ELSE
	timeoutTON.IN := FALSE;
END_IF
lastStep := step;

IF timeoutTON.Q THEN // Timeout -> Error
	errorStep:=step;
	step:=900;
END_IF


// Copy Dummy Explorervariable when Explorer Mode not used
IF ptrExplorer = 0 THEN
	ptrExplorer := ADR(explorerDummy);
	ptrExplorer^.xExecute := FALSE;
	explorerVar:=FALSE;
ELSIF ptrExplorer <> ADR(explorerDummy) THEN
	explorerVar:=TRUE;
END_IF


// Start normal send/receive Mode
IF start AND NOT lastActive AND NOT ptrExplorer^.xExecute THEN
	lastActive:=TRUE;
	STEP:=10;
ELSIF NOT start AND step=1 AND NOT ptrExplorer^.xExecute THEN
	lastActive:=FALSE;
END_IF

// Start/Stop Explorer Mode (Login/Logout)
IF ptrExplorer^.Login AND NOT lastActive THEN
	ptrExplorer^.xExecute:=TRUE;
	lastActive:=TRUE;
	step:=10;
ELSIF (ptrExplorer^.Logout OR autoLogOffTON.Q) AND ptrExplorer^.xExecute THEN
	ptrExplorer^.xExecute:=FALSE;
	lastActive:=FALSE;
	step:=90;
END_IF

//Automatic Log off
autoLogOffTON(PT:=UDINT_TO_TIME(240000)); // Automatic Logoff After 4 Minutes idle
IF step = 500 THEN // Waint for Input in WebVisu
	autoLogOffTON.IN := TRUE;
ELSE
	autoLogOffTON.IN := FALSE;
END_IF

	CASE STEP OF
	
	0:	xBusy := FALSE;
		recvComplete := FALSE;
		startSend:= FALSE;
		// Reset Connection
		ConnectionParam.MessageID[0]:=0; ConnectionParam.MessageID[1]:=0; // Reset Message ID
		ConnectionParam.MaxReadSize:= 0; ConnectionParam.MaxTransactSize:= 0; ConnectionParam.MaxWriteSize:= 0; // Reset Read/Write Size
		TCP1.ipAddr.sAddr:='0.0.0.0';
		TCP1.xEnable:= FALSE;		
		TCPRECV.xEnable:= FALSE;
		TCPSEND.xExecute:=FALSE;
		// Reset Session
		ConnectionParam.Session.SessionID[0]:= 0; ConnectionParam.Session.SessionID[1]:= 0;  // Reset Session ID
		ConnectionParam.Session.SigningRequired:=FALSE; 
		FOR i:=0 TO 15 DO
			ConnectionParam.Session.SessionKey[i]:= 0; // Reset Session Key
		END_FOR
		// Reset Tree
		ConnectionParam.Session.TreeConnect.TreeConnectId:= 0; // Reset Tree ID
		ConnectionParam.Session.TreeConnect.ShareName:= "";
		ConnectionParam.Session.TreeConnect.IsDfsShare:=FALSE;
		// Reset File
		ConnectionParam.Session.Open.FileId[0]:=0; ConnectionParam.Session.Open.FileId[1]:=0;
		ConnectionParam.Session.Open.FileId[2]:=0; ConnectionParam.Session.Open.FileId[3]:=0; // Reset File ID
		ConnectionParam.Session.Open.FileSize[0]:= 0; ConnectionParam.Session.Open.FileSize[1]:= 0; // Reset File Size
		ConnectionParam.Session.Open.ReadDataLength:=0;
		ConnectionParam.Session.Open.ReadDataOffset:=0;
		
		// Reset Explorer
		IF explorerVar THEN
			explorerMode:=FALSE;
			ptrExplorer^.busy:= TRUE;
			ptrExplorer^.xExecute:=FALSE;
			ptrExplorer^.Login:=FALSE;
			ptrExplorer^.Logout:=FALSE;
			ptrExplorer^.open:=FALSE;
			ptrExplorer^.folderUp:=FALSE;
			ptrExplorer^.folderDepth:=0;
			ptrExplorer^.online := TRUE;
			ptrExplorer^.actualsharePath:="";
			
			FOR h:=0 TO 127 DO
				ptrExplorer^.Directory[h]:= ""; // Clear all Strings
				ptrExplorer^.xdir[h]:= TRUE; 
				ptrExplorer^.xfile[h]:= TRUE; 
			END_FOR
		END_IF
		
		//Reset Functions
		readF.xExecute := FALSE;
		sendF.xExecute := FALSE;
		
		step:=1;
	
	01:	// Wait	
		
	10: // Copy Connection Parameter and etablish TCP
		xDone:=FALSE;
		ptrExplorer^.done:= TRUE;
		xBusy := TRUE;
		ptrExplorer^.busy:=FALSE;
		xError := FALSE;
		eError.Error_1 := 0;
		eError.Error_2 := 0;
		eError.TCP := 0;
		eError.ConRST := FALSE;
		ptrExplorer^.error := TRUE;
		IF ptrExplorer^.xExecute THEN // Copy Connection Settings from WebVisu
			ConnectionParam.ServerName:=ptrExplorer^.IPAdress;
			ConnectionParam.UserDomain:= ptrExplorer^.UserDomain;
			ConnectionParam.User := ptrExplorer^.User;
			ConnectionParam.Password := ptrExplorer^.Password;
			explorerMode:=TRUE;
		ELSE // Connection Setting from Input Variable
			decodeSharepath(sharePath:=ADR(SharePath),sharePathLen:=WLEN(SharePath),outSharePath:=ADR(sharePathdecoded)); // Decode Sharepath
			ConnectionParam.ServerName:=WSTRING_TO_STRING(sharePathdecoded.serverName);
			ConnectionParam.UserDomain:= Domain;
			ConnectionParam.User := User;
			ConnectionParam.Password := password;
			ConnectionParam.requestedFileName := sharePathDecoded.fileName;
		END_IF
		TCP1.ipAddr.sAddr:=ConnectionParam.ServerName;
		TCP1.xEnable:= TRUE; // Etablisch TCP Connection

	
		IF TCP1.xActive THEN // Connection etablished?
			step:= 20;
			TCPRECV.xEnable := TRUE;
		ELSIF tcp1.xError THEN
			errorStep:=step;
			step:=900;
		END_IF;
		
	20: // SMB Negotiate
		NegotiateReq(Connection:=ADR(ConnectionParam),pSend:=ADR(sendBuf[0]),pSize:=ADR(sendSize)); // Negotiate Request
		startSend:=TRUE;
		step:=30;
	
	30:	// Wait for Negotiate Response
		IF TCPSEND.xDone THEN startSend:=FALSE; END_IF; // Deactivate Send Function after successful sending#
		
		IF recvComplete AND (SMB2HeaderRep.Command = Constants.NEGOTIATE) AND (SMB2HeaderRep.Status = Constants.STATUS_SUCCESS)  THEN
			recvComplete := FALSE;
			STEP:=40;
		ELSIF recvComplete AND NOT (SMB2HeaderRep.Status = Constants.STATUS_SUCCESS) THEN
			errorStep:=step;
			step:=900;
		END_IF;
			
	40: // Session Setup, NTLMSSP Negotitate
		// Build SMB2 Header
		SMB2Header.ProtocolID[0]:= 16#FE; SMB2Header.ProtocolID[1]:= 16#53; SMB2Header.ProtocolID[2]:= 16#4D; SMB2Header.ProtocolID[3]:= 16#42; 
		SMB2Header.StructureSize := 64;
		SMB2Header.CreditCharge := 1;
		SMB2Header.Status := 0;
		SMB2Header.Command := Constants.SESSION_SETUP;
		SMB2Header.CreditRepReq := 31;
		SMB2Header.Flags:= 0;
		SMB2Header.Flags := 0;
		SMB2Header.NextCommand := 0;
		SMB2Header.MessageID[0]:= 1; SMB2Header.MessageID[1]:= 0;
		ConnectionParam.MessageID[0]:= 1;
		SMB2Header.Reserved := 0;
		SMB2Header.TreeID:= 0;
		SMB2Header.SessionID[0]:= 0; SMB2Header.SessionID[1]:= 0;
		SMB2Header.Signature[0]:= 0; SMB2Header.Signature[1]:= 0; SMB2Header.Signature[2]:= 0; SMB2Header.Signature[3]:= 0;

		// Build Session Setup Request
		SMB2SessionSetup.StructureSize:=25;
		SMB2SessionSetup.SecurityBufferOffset := SMB2Header.StructureSize + SMB2SessionSetup.StructureSize-1;
		// Build NTLM Payload
		NTLM(Connection:=ADR(ConnectionParam),pDest:=ADR(sendBuf[SMB2SessionSetup.SecurityBufferOffset+4]),Mode:= 1);
		tempLen:=INT_TO_UINT(NTLM.out);
		SMB2SessionSetup.SecurityBufferLength := tempLen;
		
		sendS:=SIZEOF(SMB2_Transport_Header);
		
		// Copy Header into Buffer
		startIndex:=sendS-1;
		sendS:=sendS+SIZEOF(SMB2_Header_Sync);
		MEM.MemMove(pSource:=ADR(SMB2Header) , pDestination:=ADR(sendBuf[startIndex]) ,uiNumberOfBytes:=SIZEOF(SMB2_Header_Sync));
		// Copy Session Setup into Buffer
		startIndex:=sendS-1;
		sendS:=sendS+SIZEOF(SMB2_SESSION_SETUP_Request);
		MEM.MemMove(pSource:=ADR(SMB2SessionSetup) , pDestination:=ADR(sendBuf[startIndex]) ,uiNumberOfBytes:=SIZEOF(SMB2_SESSION_SETUP_Request));
		// NTLMSSP
		sendS:=sendS+tempLen;
	
		// Build Transport Header
		TransportHeader.Zero := 16#00;
		TransportHeader.StreamProtocolLength := SHR(MEM.ReverseBYTEsInDWORD(sendS-SIZEOF(TransportHeader)),8); //SMB2SessionSetup.SecurityBufferLength
		
		startIndex:=0;
		MEM.MemMove(pSource:=ADR(TransportHeader) , pDestination:=ADR(sendBuf[startIndex]) ,uiNumberOfBytes:=SIZEOF(SMB2_Transport_Header)-1);
		
		sendSize:= sendS-1;
			 
		startSend:=TRUE;
		STEP:=41;
	
	41: // Wait for Session Setup Response and Challenge Message
		IF TCPSEND.xDone THEN startSend:=FALSE; END_IF; // Deactivate Send Function after successful sending
		
		IF recvComplete AND (SMB2HeaderRep.Status = Constants.STATUS_MORE_PROCESSING_REQUIRED) THEN
		recvComplete := FALSE;
		step:=42;	
		ELSIF recvComplete AND (NOT (SMB2HeaderRep.Status = Constants.STATUS_SUCCESS) OR NOT (SMB2HeaderRep.Status = Constants.STATUS_MORE_PROCESSING_REQUIRED)) THEN
			errorStep:=step;
			step:=900;
		END_IF;
		
	42:	// Compute Challenge Message
		IF ConnectionParam.LastStatus = Constants.STATUS_MORE_PROCESSING_REQUIRED THEN
			NTLM(Connection:=ADR(ConnectionParam),pDest:=ADR(recvBuf[SMB2SessionSetupRep.SecurityBufferOffset+4]),Mode:=2); // Compute Challenge Message
		END_IF
		IF NTLM.xDone THEN
			STEP:=50;
		END_IF
		
	50: // Session Setup and NTLM AUTH MESSAGE
		// Build SMB2 Header
		SMB2Header.MessageID[0]:= ConnectionParam.MessageID[0]+1; SMB2Header.MessageID[1]:= 0;
		SMB2Header.SessionID[0]:= SMB2HeaderRep.SessionID[0]; SMB2Header.SessionID[1]:= SMB2HeaderRep.SessionID[1]; 
		SMB2Header.CreditCharge := 1;
		SMB2Header.Reserved := 0;
		// Build Session Setup
		SMB2SessionSetup.StructureSize:=25;
		SMB2SessionSetup.SecurityBufferOffset := SMB2Header.StructureSize + SMB2SessionSetup.StructureSize-1;
		// Build NTLM AUTH MESSAGE Payload
		NTLM(Connection:=ADR(ConnectionParam),pSend:=ADR(sendBuf[SMB2SessionSetup.SecurityBufferOffset+4]),Mode:= 3); //Build NTLM Auth Message
		IF NTLM.xDone THEN
			ConnectionParam.MessageID[0] := ConnectionParam.MessageID[0]+1;
			step:=51;
		END_IF

	51:	// Parse Session Setup, AUTH MESSAGE to send Buffer
		tempLen:=INT_TO_UINT(NTLM.out); // Length of Security Blob
		SMB2SessionSetup.SecurityBufferLength := tempLen; // Length of Blob in Session Setup Structure
		
		// Copy Data in SendBuffer
		sendS:=SIZEOF(SMB2_Transport_Header);
		
		// SMB2 Header
		startIndex:=sendS-1;
		sendS:=sendS+SIZEOF(SMB2_Header_Sync);
		MEM.MemMove(pSource:=ADR(SMB2Header) , pDestination:=ADR(sendBuf[startIndex]) ,uiNumberOfBytes:=SIZEOF(SMB2_Header_Sync));
		// Session Setup
		startIndex:=sendS-1;
		sendS:=sendS+SIZEOF(SMB2_SESSION_SETUP_Request);
		MEM.MemMove(pSource:=ADR(SMB2SessionSetup) , pDestination:=ADR(sendBuf[startIndex]) ,uiNumberOfBytes:=SIZEOF(SMB2_SESSION_SETUP_Request));
		// Add NTLMSSP Length
		sendS:=sendS+tempLen;
	
		// Transport Header, Identifier and Length of Message
		TransportHeader.Zero := 16#00;
		TransportHeader.StreamProtocolLength := SHR(MEM.ReverseBYTEsInDWORD(sendS-SIZEOF(TransportHeader)),8); 
		
		startIndex:=0;
		MEM.MemMove(pSource:=ADR(TransportHeader) , pDestination:=ADR(sendBuf[startIndex]) ,uiNumberOfBytes:=SIZEOF(SMB2_Transport_Header)-1);
		
		sendSize:= sendS-1;
		
		startSend:=TRUE;
		step:=52;

	52:	// Wait for Session Setup / Auth Message send response	
		IF TCPSEND.xDone THEN startSend:=FALSE; END_IF; // Deactivate Send Function after successful sending
		// Wait Session Setup Reponse
		IF recvComplete AND (SMB2HeaderRep.Status = Constants.STATUS_SUCCESS) AND NOT explorerMode THEN	// Session Setup ok and read/write Mode
			recvComplete := FALSE;
			step:=61;	
		ELSIF recvComplete AND (SMB2HeaderRep.Status = Constants.STATUS_SUCCESS) AND explorerMode THEN // Session Setup ok and Explorer Mode
			recvComplete := FALSE;
			step:=520;	
		ELSIF recvComplete AND NOT (SMB2HeaderRep.Status = Constants.STATUS_SUCCESS) THEN
			errorStep:=step;
			step:=900;
		END_IF;
	
	61:	// Tree Connect	
		tempwString:=WCONCAT("\\", sharePathDecoded.serverName);
		tempwString:=WCONCAT(tempwString, "\");
		tempwString:=WCONCAT(tempwString, sharePathDecoded.treeName); // Copy \\ServerName\TreeName
	
		TreeConnectReq(Connection:=ADR(ConnectionParam),pSend:=ADR(sendBuf[0]),pSize:=ADR(sendSize),SharePathName:=tempwString); // Tree Connect Request

		startSend:=TRUE;
		step:=63;

	63:	// Wait for Tree Connect Reponse
		IF TCPSEND.xDone THEN startSend:=FALSE; END_IF; // Deactivate Send Function after successful sending
		
		IF recvComplete AND (SMB2HeaderRep.Status = Constants.STATUS_SUCCESS) THEN // Tree Connect ok
			recvComplete := FALSE;
			IF write_read = 1 THEN  // Write File to Server
				step:=220;
			ELSIF write_read = 2 THEN // Read File from Server
				step:=200;
			ELSE
				step:=900;
			END_IF
		ELSIF recvComplete AND NOT (SMB2HeaderRep.Status = Constants.STATUS_SUCCESS) THEN
			errorStep:=step;
			step:=900;
		END_IF
		
	90: // File Close on Server
		IF (ConnectionParam.Session.Open.FileId[0] <> 0) OR (ConnectionParam.Session.Open.FileId[1] <> 0)
			OR (ConnectionParam.Session.Open.FileId[2] <> 0) OR (ConnectionParam.Session.Open.FileId[3] <> 0) THEN // File Open?
			
			CloseReq(Connection:=ADR(ConnectionParam),pSend:=ADR(sendBuf[0]),pSize:=ADR(sendSize)); // Close Request
			startSend:=TRUE;
			step:=91;
		ELSE
			step:=92;
		END_IF

	91:	// Wait for File Close Response
		IF TCPSEND.xDone THEN startSend:=FALSE; END_IF; // Deactivate Send Function after successful sending
		
		IF recvComplete AND (SMB2HeaderRep.Status = Constants.STATUS_SUCCESS) THEN // Close Reques ok
			recvComplete := FALSE;
			step:= 92;
		ELSIF recvComplete AND NOT (SMB2HeaderRep.Status = Constants.STATUS_SUCCESS) THEN
			errorStep:=step;
			step:=900;
		END_IF

	92: // Tree Disconnect Request
		IF (ConnectionParam.Session.TreeConnect.TreeConnectId <> 0)  THEN // Tree connected?
			TreeDisconnectReq(Connection:=ADR(ConnectionParam),pSend:=ADR(sendBuf[0]),pSize:=ADR(sendSize)); // Tree Disconnect Request
			startSend:=TRUE;
			step:=93;
		ELSE
			step:=94;
		END_IF
	93:	// Wait for Tree Disconnect
		IF TCPSEND.xDone THEN startSend:=FALSE; END_IF; // Deactivate Send Function after successful sending
		
		IF recvComplete AND (SMB2HeaderRep.Status = Constants.STATUS_SUCCESS) THEN // Tree Disconnect Request ok
			recvComplete := FALSE;
			step:= 94;
		ELSIF recvComplete AND NOT (SMB2HeaderRep.Status = Constants.STATUS_SUCCESS) THEN
			errorStep:=step;
			step:=900;
		END_IF

	94: // Session Logoff Request
		IF (ConnectionParam.Session.SessionID[0] <> 0) OR (ConnectionParam.Session.SessionID[1] <> 0)  THEN // Session connected?
			LogOffReq(Connection:=ADR(ConnectionParam),pSend:=ADR(sendBuf[0]),pSize:=ADR(sendSize)); // LogOff Request
			startSend:=TRUE;
			step:=95;
		ELSE
			step:=0;
		END_IF
	95:	// Wait for Session Logoff Response
		IF TCPSEND.xDone THEN startSend:=FALSE; END_IF; // Deactivate Send Function after successful sending
		
		IF recvComplete AND (SMB2HeaderRep.Status = Constants.STATUS_SUCCESS) THEN // LogOff Request ok
			recvComplete := FALSE;
			xDone:= TRUE;
			ptrExplorer^.done:= FALSE;
			step:= 0;
		ELSIF recvComplete AND NOT (SMB2HeaderRep.Status = Constants.STATUS_SUCCESS) THEN
			errorStep:=step;
			step:=900;
		END_IF

	
	(* READ FILE FROM SERVER *)	
	200: // Read File
		readF(Connection:=ADR(ConnectionParam),pSend:=ADR(sendBuf[0]),pRecv:=ADR(recvBuf[0]),pSize:=ADR(sendSize),filePath:=plcFilePath,bufferSize:=BufferSize); // Read File from Server Routine
		readF.xExecute := TRUE;
		readF.received := FALSE;
		IF readF.xError THEN // readF error -> reset
			readF.xExecute:=FALSE;
			errorStep:=step;
			step:=900;
		END_IF
		IF readF.send THEN // Send next Request
			sendF.nextRound:=FALSE;
			startSend:=TRUE;
			step:=201;
		ELSIF readF.xDone THEN // Read file from server done
			readF.xExecute:=FALSE;
			step:=90;
		END_IF
		
	201:
		IF TCPSEND.xDone THEN startSend:=FALSE; END_IF; // Deactivate Send Function after successful sending
	
		IF recvComplete AND NOT readF.xDone AND (SMB2HeaderRep.Status = Constants.STATUS_SUCCESS) THEN // Read Request ok
			recvComplete := FALSE;
			readF.received := TRUE;
			readF.nextRound:=TRUE;
			step:=200;
		ELSIF recvComplete AND NOT (SMB2HeaderRep.Status = Constants.STATUS_SUCCESS) THEN
			readF.xExecute:=FALSE;
			errorStep:=step;
			step:=900;
		END_IF
	
	(* SEND FILE TO SERVER *)
	220: // Send File 
		sendF(Connection:=ADR(ConnectionParam),pSend:=ADR(sendBuf[0]),pSize:=ADR(sendSize),filePath:=plcFilePath,bufferSize:=BufferSize); // Send File to Server Routine
		sendF.xExecute := TRUE;
		IF sendF.xError THEN
			sendF.xExecute:=FALSE;
			errorStep:=step;
			step:=900;
		END_IF
		IF sendF.send THEN // Send next bytes of file
			sendF.nextRound:=FALSE;
			startSend:=TRUE;
			step:=221;
		ELSIF sendF.xDone THEN // send file to Server done
			sendF.xExecute:=FALSE;
			step:=90;
		END_IF
	221:	
		IF TCPSEND.xDone THEN startSend:=FALSE; END_IF; // Deactivate Send Function after successful sending
		
		IF recvComplete AND NOT sendF.xDone AND (SMB2HeaderRep.Status = Constants.STATUS_SUCCESS) THEN // Send Request ok
			recvComplete := FALSE;
			sendF.nextRound:=TRUE;
			step:=220;
		ELSIF recvComplete AND NOT (SMB2HeaderRep.Status = Constants.STATUS_SUCCESS) THEN 
			readF.xExecute:=FALSE;
			errorStep:=step;
			step:=900;
		END_IF
	
	(* EXPLORER MODE *)
	500: // ShareName or Directory, Wait for next Input from WebVisu
		ptrExplorer^.online := FALSE;
		
	IF ptrExplorer^.open THEN // Open Folder Button
		ptrExplorer^.open := FALSE; // Reset Open Button
		
		IF ptrExplorer^.folderDepth = 0 THEN // Acutal Sharename?
			ptrExplorer^.actualsharePath:= WCONCAT("\\" , ConnectionParam.wServerName); // concat servername to "\\"
		END_IF
		
		ptrExplorer^.actualsharePath:= WCONCAT(ptrExplorer^.actualsharePath, "\"); // "\" after actual sharepath
		ptrExplorer^.actualsharePath:= WCONCAT(ptrExplorer^.actualsharePath, ptrExplorer^.Directory[ptrExplorer^.openIndex]); // Concat Actual Share Path with choosed Folder
		
		decodeSharepath(sharePath:=ADR(ptrExplorer^.actualsharePath),sharePathLen:=WLEN(ptrExplorer^.actualsharePath),outSharePath:=ADR(ptrExplorer^.sharePathDecoded)); // Decode Sharepath for Tree Connect
		ptrExplorer^.folderDepth:= ptrExplorer^.folderDepth+1; // increase folder depth
		step:=510;
		
	ELSIF  ptrExplorer^.folderUp THEN // Folder up
		ptrExplorer^.folderUp:=FALSE;
		IF ptrExplorer^.folderDepth > 0 THEN // Check Folder depth
			ptrExplorer^.folderDepth:= ptrExplorer^.folderDepth-1;
		ELSE
			ptrExplorer^.folderDepth:= 0;
		END_IF
		
		IF ptrExplorer^.folderDepth > 0 THEN // If not lowest folder, delete last folder from Sharepath
			i:= WLEN(ptrExplorer^.actualsharePath);
			pWord := ADR(ptrExplorer^.actualsharePath);
			FOR i:=i TO 0 BY -1 DO
				IF pWord^[i] = 16#005C THEN // Search last Backslash
					pWord^[i] := 16#0000; // Terminate String
					EXIT; // Exit for
				END_IF
			END_FOR
			decodeSharepath(sharePath:=ADR(ptrExplorer^.actualsharePath),sharePathLen:=WLEN(ptrExplorer^.actualsharePath),outSharePath:=ADR(ptrExplorer^.sharePathDecoded)); // Decode Sharepath for Tree Connect
			step:=510; // Routine for Query Dir and Files
		ELSE
			step:=520; // Routine for Query Shared Folder
		END_IF
	ELSIF  ptrExplorer^.apply THEN // Routine to copy actual Sharepath to automatic SharePath
		ptrExplorer^.apply := FALSE;
		
		decodeSharepath(sharePath:=ADR(ptrExplorer^.actualsharePath),sharePathLen:=WLEN(ptrExplorer^.actualsharePath),outSharePath:=ADR(ptrExplorer^.sharePathDecoded)); // Decode Sharepath
		
		ptrExplorer^.copysharePath:= WCONCAT("\\", STRING_TO_WSTRING(ptrExplorer^.IPAdress));
		ptrExplorer^.copysharePath:= WCONCAT(ptrExplorer^.copysharePath, "\"); 
		ptrExplorer^.copysharePath:= WCONCAT(ptrExplorer^.copysharePath, ptrExplorer^.sharePathDecoded.treeName); 
		ptrExplorer^.copysharePath:= WCONCAT(ptrExplorer^.copysharePath, "\"); 
		ptrExplorer^.copysharePath:= WCONCAT(ptrExplorer^.copysharePath, ptrExplorer^.sharePathDecoded.fileName); // ConCat IP Adresse, TreeName, and actual Folder/filename
		
		IF ptrExplorer^.sharePathDecoded.fileName <> "" THEN
			ptrExplorer^.copysharePath:= WCONCAT(ptrExplorer^.copysharePath, "\"); 
		END_IF
		
		ptrExplorer^.copysharePath:= WCONCAT(ptrExplorer^.copysharePath, ptrExplorer^.Directory[ptrExplorer^.applyIndex]); // Concat choosed Filename	
	END_IF
		
		// Connect to Shared Folder
	510: // Tree Connect
		recvComplete := FALSE;
		tempwString:=WCONCAT("\\", ptrExplorer^.sharePathDecoded.serverName);
		tempwString:=WCONCAT(tempwString, "\");
		tempwString:=WCONCAT(tempwString, ptrExplorer^.sharePathDecoded.treeName); // "\\ServerName\TreeName
		TreeConnectReq(Connection:=ADR(ConnectionParam),pSend:=ADR(sendBuf[0]),pSize:=ADR(sendSize),SharePathName:=tempwString); // Tree Connect Request
		startSend:=TRUE;
		step:=511;

	511:// Tree Connect Reponse
		IF TCPSEND.xDone THEN startSend:=FALSE; END_IF; // Deactivate Send Function after successful sending
		
		IF recvComplete AND (SMB2HeaderRep.Status = Constants.STATUS_SUCCESS) THEN // Tree Connect ok
			recvComplete := FALSE;
			step:= 512;
		ELSIF recvComplete AND NOT (SMB2HeaderRep.Status = Constants.STATUS_SUCCESS) THEN
			errorStep:=step;
			step:=900;
		END_IF
	
	512: // Create Request Explorer Mode 
		CreateReq(Connection:=ADR(ConnectionParam),pSend:=ADR(sendBuf[0]),pSize:=ADR(sendSize),fileName:=ptrExplorer^.sharePathDecoded.fileName,mode:=3); // Create Request with empty Filename
		startSend:=TRUE;
		step:=513;
		
	513: // Create Response Explorer Mode
		IF TCPSEND.xDone THEN startSend:=FALSE; END_IF; // Deactivate Send Function after successful sending
		
		IF recvComplete AND (SMB2HeaderRep.Status = Constants.STATUS_SUCCESS) THEN // Create Request ok
			recvComplete := FALSE;
			step:= 514;
		ELSIF recvComplete AND NOT (SMB2HeaderRep.Status = Constants.STATUS_SUCCESS) THEN
			errorStep:=step;
			step:=900;
		END_IF
		
	514: // Query Directory Information (List of Dir and Files)
		QueryDirReq(Connection:=ADR(ConnectionParam),pSend:=ADR(sendBuf[0]),pSize:=ADR(sendSize)); // Query Directory Request (for Dir and Filenames)
		startSend:=TRUE;
		step:=515;
		
	515: // Query Directory Information Response (List of Dir and Files)
		IF TCPSEND.xDone THEN startSend:=FALSE; END_IF; // Deactivate Send Function after successful sending
		
		IF recvComplete AND (SMB2HeaderRep.Status = Constants.STATUS_SUCCESS) AND (SMB2HeaderRep.Command = Constants.QUERY_DIRECTORY) THEN // Query Directory Request ok
			recvComplete := FALSE;
			step:= 516;
		ELSIF recvComplete AND NOT (SMB2HeaderRep.Status = Constants.STATUS_SUCCESS) THEN
			errorStep:=step;
			step:=900;
		END_IF
	
	516: // Read all File names and Directory names 
		varPtr := ADR(recvBuf);
		tempOffset:=0;
		
		FOR h:=0 TO 127 DO
			ptrExplorer^.Directory[h]:= ""; // Clear all Strings
			ptrExplorer^.xdir[h]:= TRUE; // Make Buttons in WebVisu invisible
			ptrExplorer^.xfile[h]:= TRUE;  // Make Buttons in WebVisu invisible
		END_FOR
	
		j:= 0;
		// Get all Directory Names
		WHILE ((tempOffset+i) <= DWORD_TO_DINT(SMB2QueryDirRep.OutputBufferLength)) DO
			// Copy File/Dir Infofield
			MEM.MemMove(pSource:=ADR(recvBuf[SMB2QueryDirRep.OutputBufferOffset+4+tempOffset]) , pDestination:=ADR(tmpFileDirectoryInfo) ,uiNumberOfBytes:=SIZEOF(tmpFileDirectoryInfo));
			// Copy FileName from temp Infofield
			stringPtr:=ADR(ptrExplorer^.Directory[j]);
			
			IF (tmpFileDirectoryInfo.FileAtr AND 16#00000010) > 0 THEN // File Attribute = Directory?
				FOR i:=0 TO DWORD_TO_INT(tmpFileDirectoryInfo.FileNameLength) DO
				stringPtr^[i]:=varPtr^[SMB2QueryDirRep.OutputBufferOffset+4+tempOffset+SIZEOF(tmpFileDirectoryInfo)+i]; // Copy all Character
				END_FOR
				stringPtr^[i-1]:= 0; stringPtr^[i]:= 0; // Terminate wString	
				IF ptrExplorer^.Directory[j] <> "." AND ptrExplorer^.Directory[j] <> ".." THEN // if Dirname not .. and not . make Open Buttin visible in WebVisu
					ptrExplorer^.xdir[j]:= FALSE; //  False = Enable Open Button in HMI
					ptrExplorer^.xfile[j]:= TRUE; // True = Disable Apply Button in HMI
				END_IF
				
				j:=j+1;
			END_IF

			tempOffset:=tempOffset+DWORD_TO_DINT(tmpFileDirectoryInfo.NextOffset); // Offset for Next Name
			
			// Last Element Offset = 0
			IF (tmpFileDirectoryInfo.NextOffset = 0) OR (tempOffset+i >= DWORD_TO_DINT(SMB2QueryDirRep.OutputBufferLength)) THEN
				EXIT;
			END_IF
			
		END_WHILE
		
		// Get all File Names
		tempOffset:=0;
		
		WHILE ((tempOffset+i) <= DWORD_TO_DINT(SMB2QueryDirRep.OutputBufferLength)) DO
				// Copy File/Dir Infofield
				MEM.MemMove(pSource:=ADR(recvBuf[SMB2QueryDirRep.OutputBufferOffset+4+tempOffset]) , pDestination:=ADR(tmpFileDirectoryInfo) ,uiNumberOfBytes:=SIZEOF(tmpFileDirectoryInfo));
				// Copy FileName from temp Infofield
				stringPtr:=ADR(ptrExplorer^.Directory[j]);
				
				IF (tmpFileDirectoryInfo.FileAtr AND 16#00000010) = 0 THEN // File Attribute = 0 for File
					FOR i:=0 TO DWORD_TO_INT(tmpFileDirectoryInfo.FileNameLength) DO
					stringPtr^[i]:=varPtr^[SMB2QueryDirRep.OutputBufferOffset+4+tempOffset+SIZEOF(tmpFileDirectoryInfo)+i]; // Copy all Character
					END_FOR
					stringPtr^[i-1]:= 0; stringPtr^[i]:= 0; // Terminate wString	
					ptrExplorer^.xdir[j]:= TRUE; // True = Disable Open Button in HMI
					ptrExplorer^.xfile[j]:= FALSE; // False = Enable Apply Button in HMI
					j:=j+1;
				END_IF
	
				tempOffset:=tempOffset+DWORD_TO_DINT(tmpFileDirectoryInfo.NextOffset); // Offset for Next Name
				
				// Last Element Offset = 0
				IF (tmpFileDirectoryInfo.NextOffset = 0) OR (tempOffset+i >= DWORD_TO_DINT(SMB2QueryDirRep.OutputBufferLength)) THEN
					EXIT;
				END_IF
				
		END_WHILE
		step:= 550;
		
	
	
	(* NetShares *)
	(* Find all NetShare Names and hidden NetShares *)
	(* This routine is copied from Wireshark - no documentary found *)
	(* 1. Create Request "srvsvc" 2. NetShareBind 3. Read Request 4. NetShareEnumAll 5. Close Request *)
	
	520: // Tree Connect
		ptrExplorer^.actualsharePath:= WCONCAT("\\" , ConnectionParam.wServerName); // concat servername to "\\"
		ptrExplorer^.actualsharePath:= WCONCAT(ptrExplorer^.actualsharePath , "\IPC$$"); // concat IPC$
		recvComplete := FALSE;
		TreeConnectReq(Connection:=ADR(ConnectionParam),pSend:=ADR(sendBuf[0]),pSize:=ADR(sendSize),SharePathName:=ptrExplorer^.actualsharePath); // Tree Connect Request with IPC$ path
		startSend:=TRUE;
		step:=521;

	521:// Tree Connect Reponse
		IF TCPSEND.xDone THEN startSend:=FALSE; END_IF; // Deactivate Send Function after successful sending
		
		IF recvComplete AND (SMB2HeaderRep.Status = Constants.STATUS_SUCCESS) THEN // Tree Connect Request ok
			recvComplete := FALSE;
			step:= 522;
		ELSIF recvComplete AND NOT (SMB2HeaderRep.Status = Constants.STATUS_SUCCESS) THEN
			errorStep:=step;
			step:=900;
		END_IF
	
	522: // Create Request "srvsvc"
		CreateReq(Connection:=ADR(ConnectionParam),pSend:=ADR(sendBuf[0]),pSize:=ADR(sendSize),fileName:="srvsvc",mode:=4); // Create Request with srvsvc Server Service
		startSend:=TRUE;
		step:=523;	
		
	523: // Create Response "srvsvc"
		IF TCPSEND.xDone THEN startSend:=FALSE; END_IF; // Deactivate Send Function after successful sending
		
		IF recvComplete AND (SMB2HeaderRep.Status = Constants.STATUS_SUCCESS) THEN // Create Request ok
			recvComplete := FALSE;
			step:= 524;
		ELSIF recvComplete AND NOT (SMB2HeaderRep.Status = Constants.STATUS_SUCCESS) THEN
			errorStep:=step;
			step:=900;
		END_IF
	
	524: // NetShareBind 
		NetShareBind(Connection:=ADR(ConnectionParam),pSend:=ADR(sendBuf[0]),pSize:=ADR(sendSize)); // NetShareBind
		startSend:=TRUE;
		step:=525;
		
	525: // NetShareBind
		IF TCPSEND.xDone THEN startSend:=FALSE; END_IF; // Deactivate Send Function after successful sending
		
		IF recvComplete AND (SMB2HeaderRep.Status = Constants.STATUS_SUCCESS) THEN // NetShareBind ok
			recvComplete := FALSE;
			step:= 526;
		ELSIF recvComplete AND NOT (SMB2HeaderRep.Status = Constants.STATUS_SUCCESS) THEN
			errorStep:=step;
			step:=900;
		END_IF
		
	526: // NetShareBind Read - Reads the Bind
		ReadRequest(Connection:=ADR(ConnectionParam),pSend:=ADR(sendBuf[0]),pSize:=ADR(sendSize),numBytes:=1024); // Read NetShareBind
		startSend:=TRUE;
		step:=527;
		
	527: // Wait for NetShareBind Read Response
		IF TCPSEND.xDone THEN startSend:=FALSE; END_IF; // Deactivate Send Function after successful sending
		
		IF recvComplete AND (SMB2HeaderRep.Status = Constants.STATUS_SUCCESS) THEN // Read NetShareBind ok
			recvComplete := FALSE;
			step:= 528;
		ELSIF recvComplete AND NOT (SMB2HeaderRep.Status = Constants.STATUS_SUCCESS) THEN
			errorStep:=step;
			step:=900;
		END_IF	
	
	528: // NetShareEnumAll
		NetShareEnumAll(Connection:=ADR(ConnectionParam),pSend:=ADR(sendBuf[0]),pSize:=ADR(sendSize)); // NetshareEnumAll Request for shared Folder names
		startSend:=TRUE;
		step:=529;
		
	529: // Wait for NetShareEnumAll Response
		IF TCPSEND.xDone THEN startSend:=FALSE; END_IF; // Deactivate Send Function after successful sending
		
		IF recvComplete AND (SMB2HeaderRep.Status = Constants.STATUS_SUCCESS) THEN // NetshareEnumAll ok
			recvComplete := FALSE;
			step:= 530;
		ELSIF recvComplete AND NOT (SMB2HeaderRep.Status = Constants.STATUS_SUCCESS) THEN
			errorStep:=step;
			step:=900;
		END_IF
	
	530: // Decode NetShare Names
		i:= 16#04 + 16#0040 + 16#30 + 16#20 + 16#30; // Skip Transportheader + SMB2 Header + Ioctl Reponse + DCE/RPC to first Name + Number of Shares
		
		// Looking for Number < 256 - this is the first name
		FOR i:=i TO 1024 BY 8 DO
			pLWORD:=ADR(tempLWORD);
			FOR j:=0 TO 7 DO
				pLWORD^[j] := recvbuf[i+j]; // Copy 8 Byte into temp
			END_FOR;
			
			IF (tempLWORD < 256) AND (tempLWORD > 0) THEN // Check temp for Number < 256 and > 0, then this ist the Length of first Name
				EXIT;
			END_IF
		END_FOR;
		
		FOR h:=0 TO 127 DO
			ptrExplorer^.Directory[h]:= ""; // Clear all Strings
			ptrExplorer^.xdir[h]:= TRUE;  // Make Open Button invisible in WebVisu
			ptrExplorer^.xfile[h]:= TRUE; // Make apply Button invisible in WebVisu
		END_FOR
		h:=0;
		numberOfNames:=0;
		// This decodes the NetShareEnumAll Reponse. I found no doc for that
		// first name ist the sharename followed by an emtpy string or if it not emtpy it is the commentary for the share.
		
		WHILE (h<=127) AND i <= UDINT_TO_DINT(BufferSize)-1 AND i>0  DO
			// Decode first Name - 2 LWORD of Length with Zero LWORD between
			pLWORD:=ADR(tempLWORD); // First Length (Max Length?)
			FOR j:=0 TO 7 DO
				pLWORD^[j] := recvbuf[i+j]; // Copy 8 Byte of first Length
			END_FOR;
			i:=i+2*8; // Empty 8 Bytes
			pLWORD:=ADR(tempLWORD2); // Second Length (Actual Length?)
			FOR j:=0 TO 7 DO
				pLWORD^[j] := recvbuf[i+j]; // Copy 8 Byte of second Length
			END_FOR;
			i:=i+8;
			
			// If the two Length Match than decode the Name
			IF tempLWORD = tempLWORD2 THEN 
				pVar := ADR(ptrExplorer^.Directory[h]);
				tempLWORD := tempLWORD + tempLWORD; // Double the Length. Length = Characters but WSTRING needs 2 byte for 1 Char
				IF (tempLWORD MOD 8) > 0 THEN
					tempLWORD := tempLword+(8-(tempLWORD MOD 8)); // Length + padding bytes 
				END_IF
				FOR j:=0 TO LWORD_TO_INT(tempLWORD) DO // Copy Name into WString
					pVar^[j] := recvbuf[i+j];
				END_FOR
				IF (numberOfNames MOD 2) = 0 THEN // Don't increase index after second string - commentary
					h:=h+1;	// Index for List
				END_IF
				numberOfNames := numberOfNames + 1; // Number of decoded Strings
			END_IF
			i:=i+LWORD_TO_INT(tempLWORD); // i+ Length of Name for start of next Length/Name
		END_WHILE
		
		// Make Open Button visible in Explorer
		FOR i:=0 TO 127 DO
			IF (WLEN(ptrExplorer^.Directory[i]) > 0) THEN // Open Button visible for all shared Folders
				ptrExplorer^.xdir[i]:= FALSE;
			END_IF
		END_FOR
		
		step:= 550;
	

		
	550: // File Close Request - After NetShare or Query Directory
		IF (ConnectionParam.Session.Open.FileId[0] <> 0) OR (ConnectionParam.Session.Open.FileId[1] <> 0)
			OR (ConnectionParam.Session.Open.FileId[2] <> 0) OR (ConnectionParam.Session.Open.FileId[3] <> 0) THEN // File Open?
			CloseReq(Connection:=ADR(ConnectionParam),pSend:=ADR(sendBuf[0]),pSize:=ADR(sendSize)); // File Close Request
			startSend:=TRUE;
			step:=551;
		ELSE
			step:=552; // File already closed
		END_IF
		
	551: // Wait File Close Response
		IF TCPSEND.xDone THEN startSend:=FALSE; END_IF; // Deactivate Send Function after successful sending

		IF recvComplete AND (SMB2HeaderRep.Status = Constants.STATUS_SUCCESS) THEN // File Close Request ok?
			recvComplete := FALSE;
			step:= 552;
		ELSIF recvComplete AND NOT (SMB2HeaderRep.Status = Constants.STATUS_SUCCESS) THEN
			errorStep:=step;
			step:=900;
		END_IF
		
	552: // Tree Disconnect Request
		IF (ConnectionParam.Session.TreeConnect.TreeConnectId <> 0)  THEN // Tree connected?
			TreeDisconnectReq(Connection:=ADR(ConnectionParam),pSend:=ADR(sendBuf[0]),pSize:=ADR(sendSize)); // Tree Disconnect Request
			startSend:=TRUE;
			step:=553;
		ELSE
			step:=500; // Tree already disconnected
		END_IF
	553: // Wait for Tree Disconnect Response
		IF TCPSEND.xDone THEN startSend:=FALSE; END_IF; // Deactivate Send Function after successful sending
		
		IF recvComplete AND (SMB2HeaderRep.Status = Constants.STATUS_SUCCESS) THEN // Tree Disconnect ok
			recvComplete := FALSE;
			step:= 500;
		ELSIF recvComplete AND NOT (SMB2HeaderRep.Status = Constants.STATUS_SUCCESS) THEN
			errorStep:=step;
			step:=900;
		END_IF
	
	
	// Error Handling
	900:	eError.Error_1:=errorStep;	// Copy Stepnumber
			eError.Error_2:=SMB2HeaderRep.Status; // Copy SMB2 Error
			eError.TCP:=TCP1.eError;
			
			xError := TRUE;
			
			ptrExplorer^.error := FALSE; // Indicator WebVisu
			
			step:=0;
		

	END_CASE;
	
	// RECEIVE FROM SERVER
	IF startSend THEN
		TCPRECV.xEnable:=TRUE; // Enable Send Function
	END_IF	
	
	TCP1( udiTimeOut:= (timeout*1000), uiPort:=445, eError=>Erro, xActive=>active,hConnection=>hCon ); (* TCP Client *)
	TCPSEND( xExecute:=startSend AND TCP1.xActive, hConnection:=hCon, pData:=ADR(sendBuf), szSize:=sendSize); (* TCP Write function *)
	
	IF TCPSEND.xDone THEN // Reset for receive if Send Done
		MessageLength:= 0;
		newBufferIndex:= 0;
		recvLength:=0;
	END_IF
	
	TCPRECV(hConnection:=hCon,xEnable:=TCP1.xActive, szSize:=SIZEOF(recvBuf)-recvLength, pData:=ADR(recvBuf[newBufferIndex])); (* TCP Receive function *)
	
	IF TCPRECV.xReady THEN // After every received Packet check for fragmented Packets
		
		IF MessageLength = 0 THEN // IF Message Length already decoded then don't decode again
			// TRANSPORT HEADER - Read Length of whole message from Transport Header and validate
			repP := ADR(TransportHeaderRep);
			FOR repIndex:=0 TO 3 DO // Copy header from buffer to struct
				repP^ := recvBuf[repIndex];
				repP := repP + 1;
			END_FOR	
			
			MessageLength := DINT_TO_UDINT(SHR(MEM.ReverseBYTEsInDWORD(TransportHeaderRep.StreamProtocolLength),8) AND 16#00FFFFFF)+4; // Network Byte Order to Little Endian and Shft (Length in Header 3 Byte, UDINT = 4 Byte)
		END_IF
		
		// First check if new Data match
		IF (MessageLength <> TCPRECV.szCount) AND (MessageLength <> recvLength) THEN
			recvLength:= recvLength + TCPRECV.szCount; // increase by received Length
			newBufferIndex:=recvLength; // Set Bufferposition to the End of Data
		END_IF
		
		// After that check if new data match
		IF (MessageLength = TCPRECV.szCount) OR (MessageLength = recvLength) THEN
			recvLength:=0;
			MessageLength:= 0;
			newBufferIndex:= 0;
			recvOK:=TRUE;
		END_IF
	END_IF	
		
	// Decode received Data into SMB2 Responses
	IF recvOK AND NOT recvComplete THEN		
		recvOK:=FALSE;
		
		// SMB2 HEADER
		repP := ADR(SMB2HeaderRep);
		FOR repIndex:=0 TO SIZEOF(SMB2_Header_Sync)-1 DO // Copy header from buffer to struct
			repP^ := recvBuf[repIndex+4];
			repP := repP + 1;
		END_FOR	
		
		// STRUCTURE SIZE OF COMMAND
		tmpIndex := repIndex;
		repP := ADR(repSize);
		repP^ := recvBuf[repIndex+4];
		repP := repP + 1; repIndex:=repIndex+1;
		repP^ := recvBuf[repIndex+4];
		// Copy Connection Information
		ConnectionParam.LastStatus := SMB2HeaderRep.Status;
			
		// NEGOTIATE RESPONSE	
		IF SMB2HeaderRep.Command = Constants.NEGOTIATE THEN
			
			repP:=ADR(SMB2NegotiateRep);
			FOR repIndex:=tmpIndex TO (RepSize-1)+tmpIndex DO
				repP^ := recvBuf[repIndex+4];
				repP := repP + 1;
			END_FOR	
		END_IF;	
		
		// SESSION SETUP RESPONSE
		IF SMB2HeaderRep.Command = Constants.SESSION_SETUP THEN
			
			repP:=ADR(SMB2SessionSetupRep);
			FOR repIndex:=tmpIndex TO (RepSize-1)+tmpIndex DO
				repP^ := recvBuf[repIndex+4];
				repP := repP + 1;
			END_FOR	
		ConnectionParam.Session.SessionID[0]:= SMB2HeaderRep.SessionID[0]; ConnectionParam.Session.SessionID[1]:= SMB2HeaderRep.SessionID[1];
		END_IF;			
		
		// Tree Connect Response
		IF SMB2HeaderRep.Command = Constants.TREE_CONNECT THEN
			repP:=ADR(SMB2TreeConnectRep);
			FOR repIndex:=tmpIndex TO (RepSize-1)+tmpIndex DO
				repP^ := recvBuf[repIndex+4];
				repP := repP + 1;
			END_FOR	
			// Copy Tree Information
			ConnectionParam.Session.TreeConnect.TreeConnectId := SMB2HeaderRep.TreeID;
			ConnectionParam.Session.TreeConnect.ShareName := SharePath;
		END_IF
		
		// Create Response
		IF SMB2HeaderRep.Command = Constants.CREATE THEN
			repP:=ADR(SMB2CreateRep);
			FOR repIndex:=tmpIndex TO (RepSize-1)+tmpIndex DO
				repP^ := recvBuf[repIndex+4];
				repP := repP + 1;
			END_FOR	
			// Copy File Information
			ConnectionParam.Session.Open.FileId:= SMB2CreateRep.FileId; // File ID
			ConnectionParam.Session.Open.FileSize:= SMB2CreateRep.EndofFile; // File Size
		END_IF
		
		// Write Response
		IF SMB2HeaderRep.Command = Constants.WRITE THEN
			repP:=ADR(SMB2WriteRep);
			FOR repIndex:=tmpIndex TO (RepSize-1)+tmpIndex-1 DO
				repP^ := recvBuf[repIndex+4];
				repP := repP + 1;
			END_FOR	
		END_IF
		
		// Read Response (without Buffer)
		IF SMB2HeaderRep.Command = Constants.READ THEN
			repP:=ADR(SMB2ReadRep);
			FOR repIndex:=tmpIndex TO (RepSize-1)+tmpIndex-1 DO
				repP^ := recvBuf[repIndex+4];
				repP := repP + 1;
			END_FOR	
			// Copy Read Information
			ConnectionParam.Session.Open.ReadDataOffset:= SMB2ReadRep.DataOffset; // Data Offset from Start of File
			ConnectionParam.Session.Open.ReadDataLength:= SMB2ReadRep.DataLength; // Length of Data
		END_IF
		
		// Close Response
		IF SMB2HeaderRep.Command = Constants.CLOSE THEN
			repP:=ADR(SMB2CloseRep);
			FOR repIndex:=tmpIndex TO (RepSize-1)+tmpIndex-1 DO
				repP^ := recvBuf[repIndex+4];
				repP := repP + 1;
			END_FOR	
			// Delete File ID
			FOR i:=0 TO 3 DO
				ConnectionParam.Session.Open.FileId[i]:= 0; // File ID
			END_FOR
			ConnectionParam.Session.Open.FileSize[0]:= 0; ConnectionParam.Session.Open.FileSize[1]:= 0;// File Size
		END_IF
		
		// Tree Disconnect Response
		IF SMB2HeaderRep.Command = Constants.TREE_DISCONNECT THEN
			repP:=ADR(SMB2DisconnectRep);
			FOR repIndex:=tmpIndex TO (RepSize-1)+tmpIndex-1 DO
				repP^ := recvBuf[repIndex+4];
				repP := repP + 1;
			END_FOR	
			// Delete Tree ID
			ConnectionParam.Session.TreeConnect.TreeConnectId:= 0; // File ID
			ConnectionParam.Session.TreeConnect.ShareName := "";
			ConnectionParam.Session.TreeConnect.IsDfsShare:=FALSE;
		END_IF
		
		// Logoff Response
		IF SMB2HeaderRep.Command = Constants.LOGOFF THEN
			repP:=ADR(SMB2LogoffRep);
			FOR repIndex:=tmpIndex TO (RepSize-1)+tmpIndex-1 DO
				repP^ := recvBuf[repIndex+4];
				repP := repP + 1;
			END_FOR	
			// Delete Session ID
			ConnectionParam.Session.SessionID[0] := 0; ConnectionParam.Session.SessionID[1] := 0; // Session ID
		END_IF
		
		// Query Directory Response
		IF SMB2HeaderRep.Command = Constants.QUERY_DIRECTORY THEN
			repP:=ADR(SMB2QueryDirRep);
			FOR repIndex:=tmpIndex TO (RepSize-1)+tmpIndex-1 DO
				repP^ := recvBuf[repIndex+4];
				repP := repP + 1;
			END_FOR	
		END_IF
		
		recvComplete := TRUE;
		recvP:=ADR(recvBuf);
	END_IF

END_FUNCTION_BLOCK

// Device/Application/Bausteine/SMB2_Client/SMB2/Functions/decodeSharePath
FUNCTION decodeSharePath : int
VAR_INPUT
	sharePath:POINTER TO ARRAY[0..1024] OF WORD; // Pointer Complete Sharepath
	sharePathLen:INT; // Length of Sharepath
	outSharePath:POINTER TO sharePath; // Decoded share Path
END_VAR
VAR
	pVar:POINTER TO ARRAY[0..1024] OF WORD;
	tempwString:WSTRING(512);
	i:INT;
	j:int;
END_VAR

// This Function decodes the Sharepath into Servername, Treename and Filename

i:=0;
j:=0;
//Decode ServerName
tempwString:="";
pVar := ADR(tempwString);
IF sharePath^[0] = 16#005C AND sharePath^[1] = 16#005C THEN // 16#005C = \
	i:=i+2;
	WHILE (sharePath^[i] <> 16#005C) AND NOT (i>=sharePathLen) DO // copy Name until next "\"
		pVar^[j] := sharePath^[i];
		i:=i+1;
		j:=j+1;
	END_WHILE
END_IF
pVar^[j] := 16#0000; // Terminate String
outSharePath^.serverName := tempwString;

// Decode Tree Name
j:=0;
i:=i+1;
tempwString:="";
WHILE (sharePath^[i] <> 16#005C) AND NOT (i>=sharePathLen) DO // copy Name until next "\"
	pVar^[j] := sharePath^[i];
	i:=i+1;
	j:=j+1;
END_WHILE
pVar^[j] := 16#0000; // Terminate String
outSharePath^.treeName := tempwString;

// Decode File Name
j:=0;
i:=i+1;
tempwString:="";
WHILE NOT (i>=sharePathLen) DO // copy Name end of String
	pVar^[j] := sharePath^[i];
	i:=i+1;
	j:=j+1;
END_WHILE
pVar^[j] := 16#0000; // Terminate String
outSharePath^.fileName := tempwString;

END_FUNCTION

// Device/Application/Bausteine/SMB2_Client/SMB2/Functions/Requests/NegotiateReq
FUNCTION NegotiateReq : int
VAR_INPUT
	Connection:POINTER TO Connection; // Connection Parameter
	pSend:POINTER TO ARRAY[0..32767] OF BYTE; // Pointer to Send Buffer
	pSize:POINTER TO CAA.SIZE; // Send Size
END_VAR
VAR
	TransportHeader:SMB2_Transport_Header;
	SMB2Header: SMB2_Header_Sync;
	SMBHeader: SMB_Header;
	SMBNegotiate:SMB_COM_NEGOTIATE;
	SMB2TreeConnect:SMB2_TREE_CONNECT_Request;
	sendS:UINT;
	startIndex:UINT;
END_VAR

// This Function generates the Negotiate Request (not SMB 2, its SMB1 for Negotiate)
	// SMB Negotiate
	(*Build SMB Header*)
	SMBHeader.Protocol[0]:= 16#FF; SMBHeader.Protocol[1]:= 16#53; SMBHeader.Protocol[2]:= 16#4D; SMBHeader.Protocol[3]:= 16#42;
	SMBHeader.Command := 16#72; // Negotiate
	SMBHeader.Status := 0;
	SMBHeader.Flags := Constants.SMB_FLAGS_CANONICALIZED_PATHS OR Constants.SMB_FLAGS_CASE_INSENSITIVE;
	SMBHeader.Flags2 := Constants.SMB_FLAGS2_UNICODE OR Constants.SMB_FLAGS2_NT_STATUS OR Constants.SMB_FLAGS2_IS_LONG_NAME OR Constants.SMB_FLAGS2_EAS	OR Constants.SMB_FLAGS2_LONG_NAMES;
	SMBHeader.PIDHigh:= 0;
	SMBHeader.SecurityFeatures[0] := 0;
	SMBHeader.Reserved := 0;
	SMBHeader.TID := 65535;
	SMBHeader.PIDLow := 65279;
	SMBHeader.UID := 0;
	SMBHeader.MID := 0;
	(*Build SMB_COM_NEGOTIATE*)
	SMBNegotiate.WORDCOUNT := 0;
	SMBNegotiate.Dialects[0].BufferFormat := 16#02;
	SMBNegotiate.Dialects[0].DialectString := 'SMB 2.002'; // SMB2 Version
	SMBNegotiate.BYTECOUNT := INT_TO_UINT(Len(SMBNegotiate.Dialects[0].DialectString)+1+1);
		
		
	// Copy Data in SendBuffer
	sendS:=SIZEOF(SMB2_Transport_Header);
		
	(*Parse SMB2 Header*)	
	startIndex:=sendS-1;
	sendS:=sendS+SIZEOF(SMB_Header);
	MEM.MemMove(pSource:=ADR(SMBHeader) , pDestination:=ADR(pSend^[startIndex]) ,uiNumberOfBytes:=SIZEOF(SMB_Header));
	
	(*Parse Negotiate Request*)		
	startIndex:=sendS-1;
	sendS:=sendS+WORD_TO_UINT(SMBNegotiate.BYTECOUNT)+3;
	MEM.MemMove(pSource:=ADR(SMBNegotiate) , pDestination:=ADR(pSend^[startIndex]) ,uiNumberOfBytes:=WORD_TO_UINT(SMBNegotiate.BYTECOUNT)+3);

	(*Build Header*)
	TransportHeader.Zero := 16#00;
	TransportHeader.StreamProtocolLength := SHR(MEM.ReverseBYTEsInDWORD(sendS-SIZEOF(TransportHeader)),8);
	
	startIndex:=0;
	MEM.MemMove(pSource:=ADR(TransportHeader) , pDestination:=ADR(pSend^[startIndex]) ,uiNumberOfBytes:=SIZEOF(SMB2_Transport_Header)-1);
	
	(*Set Sendsize*)	
	pSize^:= sendS-1;

END_FUNCTION

// Device/Application/Bausteine/SMB2_Client/NTLM/Functions/NTLM
FUNCTION_BLOCK NTLM
VAR_INPUT
	Connection:POINTER TO Connection; // Connection Parameter
	pDest:POINTER TO ARRAY[0..32767] OF BYTE; // Receivebuffer (for Challenge Message)
	pSend:POINTER TO ARRAY[0..32767] OF BYTE; // Send Buffer (for Negotiate and Auth Message)
	Mode:INT; // 1 = Negotiate, 2 = Process Challenge Message and Generate Auth Message, 3 = Copy Auth Message into Send Buffer and calculate MIC
	xExecute:INT; // Start
END_VAR
VAR_OUTPUT
	xDone:BOOL;
	out:int;
END_VAR
VAR
	GenerateAuthMess:GenerateAuthenticateMessage;
	step:INT;
	i:INT;
	j:int;
	pVar:POINTER TO BYTE;
	pTargN:POINTER TO ARRAY[0..32767] OF BYTE;
	pNeg:POINTER TO BYTE;
	pAuth:POINTER TO BYTE;
	NegMess:NEGOTIATE_MESSAGE;
	ChallMess:CHALLENGE_MESSAGE;
	AuthMess:AUTHENTICATE_MESSAGE;
	Session:sessionData;
	NTLMLength:UINT;
	AVList:AVPairList;
	
	OctGSS:INT;
	OctOID:INT;
	OctSPNEGO:INT;
	OctNegTokenInit:INT;
	OctContents:INT;
	OctMechTypes:INT;
	OctMechTypeNTLMSSP:INT;
	OctNTLMID:INT;
	OctNTLMObj:INT;
	OctNegTotekTarg:INT;
	DER:DER_Encoding;
	tempLen:INT;
	tempInt:INT;
	DERLen:DER_Len;
	ProcessChall:ProcessChallengeMessage;
	MIC:MIC;
END_VAR

VAR CONSTANT
	OIDLen:BYTE:=6;
	OID:ARRAY[0..OIDLen-1] OF BYTE:= [16#2B, 16#06, 16#01, 16#05, 16#05, 16#02];
	NTLMSSPLen:BYTE:=10;
	NTLMSSP:ARRAY[0..NTLMSSPLen-1] OF BYTE:= [16#2B, 16#06, 16#01, 16#04, 16#01, 16#82, 16#37, 16#02, 16#02, 16#0A];
END_VAR

pVar:=pDest;
xDone:=FALSE;

// Mode 1, Build NTLM NEGOIATE Message
	IF Mode= 1 THEN	
		NTLMLength:=SIZEOF(NEGOTIATE_MESSAGE);
		
		// Length of the Octet for every Identifier
		tempLen:=UDINT_TO_INT(SIZEOF(NEGOTIATE_MESSAGE));
		DER(Length:=tempLen, TestLen:=TRUE, NumOct=>OctNTLMID);
		tempLen:= UINT_TO_INT(SIZEOF(NEGOTIATE_MESSAGE))+OctNTLMID;
		DER(Length:=tempLen, TestLen:=TRUE, NumOct=>OctNTLMObj);
		OctMechTypeNTLMSSP:= 2;
		OctMechTypes:=2;
		OctContents:=2;
		tempLen:=UINT_TO_INT(SIZEOF(NEGOTIATE_MESSAGE))+OctNTLMID+OctNTLMObj+OctMechTypeNTLMSSP+OctMechTypes+OctContents+OIDLen+NTLMSSPLen;
		DER(Length:=tempLen, TestLen:=TRUE, NumOct=>OctNegTokenInit);
		DER(Length:=tempLen+OctNegTokenInit, TestLen:=TRUE, NumOct=>OctSPNEGO);
		OctOID:=2;
		
	
		// Start of GSS
		pVar^:= 16#60; // Start Sequence
		pVar:=pVar +1;
		// Length
		templen:=UINT_TO_INT(SIZEOF(NEGOTIATE_MESSAGE))+OctNTLMID+OctNTLMObj+OctMechTypeNTLMSSP+OctMechTypes+OctContents+OctNegTokenInit+OctSPNEGO+OctOID+OIDLen+NTLMSSPLen;
		DER(Length:=tempLen, pDest:=pVar, TestLen:=FALSE, pOut=>pVar);
		// OID
		pVar^ := 16#06; // Start Object ID
		pVar:=pVar +1;
		// Length OID
		pVar^:= OIDLen;
		pVar:=pVar +1;
		// OID
		FOR i:=0 TO OIDLen-1 DO
			pVar^:=OID[i];
			pVar:=pVar +1;
		END_FOR
		
		// SPNEGO
		pVar^:= 16#A0; //SPNEGO Start
		pVar:=pVar +1;
		// Length
		templen:=UINT_TO_INT(SIZEOF(NEGOTIATE_MESSAGE))+OctNTLMID+OctNTLMObj+OctMechTypeNTLMSSP+OctMechTypes+OctContents+OctNegTokenInit+NTLMSSPLen;
		DER(Length:=tempLen, pDest:=pVar, TestLen:=FALSE, pOut=>pVar);
		
		// NegTokenInit
		pVar^:= 16#30; //NegToken Start
		pVar:=pVar +1;
		// Length
		tempLen:=UINT_TO_INT(SIZEOF(NEGOTIATE_MESSAGE))+OctNTLMID+OctNTLMObj+OctMechTypeNTLMSSP+OctMechTypes+OctContents+NTLMSSPLen;
		DER(Length:=tempLen, pDest:=pVar, TestLen:=FALSE, pOut=>pVar);
		
		// Contents
		pVar^:= 16#A0; // Start
		pVar:=pVar +1;
		// Length
		tempLen:= NTLMSSPLen+OctMechTypeNTLMSSP+OctMechTypes;
		DER(Length:=tempLen, pDest:=pVar, TestLen:=FALSE, pOut=>pVar);
		
		// MechTypes
		pVar^:= 16#30; //MechTypes Start
		pVar:=pVar +1;
		// Length
		tempLen:= NTLMSSPLen+OctMechTypeNTLMSSP;
		DER(Length:=tempLen, pDest:=pVar, TestLen:=FALSE, pOut=>pVar);
		
		// MechType NTLMSSP
		pVar^:= 16#06; // ID
		pVar:=pVar +1;
		pVar^:= NTLMSSPLen; // Length
		pVar:=pVar +1;
		FOR i:=0 TO NTLMSSPLen-1 DO
			pVar^:=NTLMSSP[i];
			pVar:=pVar +1;
		END_FOR
		
		// NTLM ID
		pVar^:= 16#A2; // ID
		pVar:=pVar +1;
		// Length
		tempLen:=UINT_TO_INT(SIZEOF(NEGOTIATE_MESSAGE))+OctNTLMID;
		DER(Length:=tempLen, pDest:=pVar, TestLen:=FALSE, pOut=>pVar);
		
		pVar^:= 16#04; // ID
		pVar:=pVar +1;
		// Length
		tempLen:=UINT_TO_INT(SIZEOF(NEGOTIATE_MESSAGE));
		DER(Length:=tempLen, pDest:=pVar, TestLen:=FALSE, pOut=>pVar);
		
		NegMess.NegotiateFlags:= 16#E2080297;
		// Copy Negoiate Message into Buffer
		pNeg:=ADR(NegMess);
		FOR i:=0 TO tempLen-1 DO
			pVar^:= pNeg^;
			pVar:=pVar +1;
			pNeg:=pNeg +1;
		END_FOR
		
		// Copy Neg Mess for MIC
		pNeg:=ADR(NegMess);
		FOR i:=0 TO tempLen-1 DO
			session.NegMessByte[i]:= pNeg^;
			pNeg:=pNeg +1;
		END_FOR
		session.NegMessByteLen := tempLen;
		
		// Length of Security Blob
		out:= DWORD_TO_INT(pVar - pDest);
	END_IF

	// Decode Security Blob and Challenge Message, Process Challenge Message
IF Mode = 2 THEN
	CASE step OF
		0:	step:=1;
		1:	IF pVar^ = 16#A1 THEN // Start of Security Blob
					pVar:=pVar+1;
					DERLen(pSource:= pVar, pOut=> pVar,Length=>tempLen);
					// Looking for Start of CHALLENGE MESSAGE
					tempInt:= OSCAT_BASIC.BUFFER_SEARCH(PT:=pDest,SIZE:=tempLen,STR:='NTLMSSP',POS:=0,IGN:=FALSE);
					IF tempInt <> -1 THEN
						MEM.MemMove(pSource:=(pDest+INT_TO_UINT(tempInt)) , pDestination:=ADR(ChallMess) ,uiNumberOfBytes:=56); // Copy Challenege Message from Buffer in Struct
					END_IF
					
				// Target Name
				pTargN:= ADR(ChallMess.TargetName);
				FOR i:=0 TO WORD_TO_INT(ChallMess.TargetNameLen)-1 DO
					pTargN^[i] := pDest^[i+tempInt+DWORD_TO_INT(ChallMess.TargetNameBufferOffset)]; // Copy Targetname
				END_FOR	
				pTargN^[i]:= 0; pTargN^[i+1]:= 0; // String Termination
				
				// Attribute, Decode AV Pairs
				GetAVPairList(pSource:=pDest+INT_TO_DWORD(tempInt)+ChallMess.TargetInfoBufferOffset,ChallMess:=ADR(ChallMess)); // Get Attributes from Target Info
				Connection^.wServerName:= challmess.AVPairList.DNSComputerName; // Get ComputerName for ExplorerMode
				
				// Copy whole Challenge for MIC calculation
				pVar:=pDest+INT_TO_UINT(tempInt);
				FOR i:=0 TO tempLen+4-1-tempint-1 DO
					session.ChallMessByte[i] := pVar^;
					pVar:=pVar +1;
				END_FOR
				session.ChallMessByteLen := i;
				
				step:=2;
			END_IF
			
			
			// Process Challenge Message	
		2:	Session.userDomain:=Connection^.UserDomain;
			Session.user:=Connection^.User;
			Session.password:=Connection^.Password;
			ProcessChall(session:=ADR(Session),challMess:=ADR(ChallMess)); // Process the Challenge Message with all Responses and Keys
			ProcessChall.xExecute := TRUE;
			
			IF ProcessChall.xDone THEN
				step:=3;
			END_IF
			
			// Generate Auth Message
		3: 	GenerateAuthMess(session:= ADR(Session),authMess=>AuthMess);
			xDone:=TRUE;
			step:=0;
	END_CASE
END_IF	
	// Mode 3, Parse AuthMessage to Send Buffer
IF Mode = 3 THEN
	CASE step OF
		0:	step:=1;
		1: 	MIC(session:=ADR(session),out=>AuthMess.MIC); // Generate the MIC over all 3 Messages
			MIC.xExecute := TRUE;
			IF mic.xDone THEN
				MIC.xExecute := FALSE;
				step:=2;
			END_IF
		2:	pVar:= pSend;
			// NTML Message Length, Auth+Payload
			tempLen:=88+AuthMess.PayLoadSize;
			DER(Length:=tempLen, TestLen:=TRUE, NumOct=>OctNTLMID);
			// NTMLID
			tempLen:= 88+AuthMess.PayLoadSize+OctNTLMID+20;
			DER(Length:=tempLen, TestLen:=TRUE, NumOct=>OctNTLMObj);
			// negTokenTarg
			tempLen:= 88+AuthMess.PayLoadSize+OctNTLMID+OctNTLMObj+5+20;
			DER(Length:=tempLen, TestLen:=TRUE, NumOct=>OctNegTotekTarg);
			// GSS API
			tempLen:= 88+AuthMess.PayLoadSize+OctNTLMID+OctNTLMObj+5+OctNegTotekTarg+20;
			DER(Length:=tempLen, TestLen:=TRUE, NumOct=>OctSPNEGO);
			
			// GSS-API
			//	a1 - identifier
			// octect over all	
			pVar^ := 16#A1;
			pVar:=pVar+1;
			templen:=88+AuthMess.PayLoadSize+OctNTLMID+OctNTLMObj+5+OctNegTotekTarg+20;
			DER(Length:=tempLen, pDest:=pVar, TestLen:=FALSE, pOut=>pVar);
	
			// negTokenTarg
			// 30 - Identifier
			// octect over all - GSS
			pVar^ := 16#30;
			pVar:=pVar+1;
			templen:=88+AuthMess.PayLoadSize+OctNTLMID+OctNTLMObj+5+20;
			DER(Length:=tempLen, pDest:=pVar, TestLen:=FALSE, pOut=>pVar);
			
			// negResult 0a 03
			// a0	
			// length 03
			// accept-incomplete 0a 01 01
			// 0a idetifier
			// lenght 01
			// 01 - neg result accept incomplete
			pVar^:= 16#A0; // Identifier
			pVar:=pVar+1;
			pVar^:= 16#03; // Length (identifier + Length + accept incomplete)
			pVar:=pVar+1;
			pVar^:= 16#0A; // Identifier negResult
			pVar:=pVar+1;
			pVar^:= 16#01; // length negResult
			pVar:=pVar+1;
			pVar^:= 16#01; // Accept Incomplete
			pVar:=pVar+1;
			
			// a2
			// length overall + 4
			pVar^ := 16#A2;
			pVar:=pVar+1;
			templen:=88+AuthMess.PayLoadSize+OctNTLMID;
			DER(Length:=tempLen, pDest:=pVar, TestLen:=FALSE, pOut=>pVar);
			
			// 04 idenftifier for AUTH MESSAGE
			// length of AUTH_MESS
			pVar^ := 16#04;
			pVar:=pVar+1;
			templen:=88+AuthMess.PayLoadSize;
			DER(Length:=tempLen, pDest:=pVar, TestLen:=FALSE, pOut=>pVar);
			
			// Copy Auth Message into Buffer
			pAuth:=ADR(AuthMess);
			tempLen:=88;
			FOR i:=0 TO tempLen-1 DO
				pVar^:= pAuth^;
				pVar:=pVar +1;
				pAuth:=pAuth +1;
			END_FOR
			
			// Copy Auth Payload into
			pAuth:=ADR(AuthMess.Payload);
			tempLen:=88;
			FOR i:=0 TO AuthMess.PayLoadSize-1 DO
				pVar^:= pAuth^;
				pVar:=pVar +1;
				pAuth:=pAuth +1;
			END_FOR
			
			// Copy mechListMIC
			FOR i:=0 TO 19 DO
				pVar^ := session.mechListMIC[i];
				pVar:=pVar +1;
			END_FOR
			
			// Length of Security Blob for SMB Message
			out:= DWORD_TO_INT(pVar - pSend);
			xDone:=TRUE;
			step:=0;
	END_CASE
END_IF

END_FUNCTION_BLOCK

// Device/Application/Bausteine/SMB2_Client/NTLM/Functions/MIC
FUNCTION_BLOCK MIC
VAR_INPUT
	xExecute:BOOL;
	session:POINTER TO SessionData;
END_VAR
VAR_OUTPUT
	out:ARRAY[0..15] OF BYTE;
	xDone:BOOL;
END_VAR
VAR
	step:int:=0;
	temp:ARRAY[0..2048] OF BYTE;
	j:INT;
	i:INT;
	HMACMD5:HMAC_MD5;
END_VAR

// This Function generates the MIC over all 3 Messages
//MIC=HMAC_MD5(ExportedSessionKey,ConcatenationOf(NEGOTIATE_MESSAGE,CHALLENGE_MESSAGE,AUTHENTICATE_MESSAGE)):
xDone := FALSE;
IF Step = 0 AND xExecute = 1 THEN
	Step:=1;
END_IF
CASE step OF
	// ConcatenationOf(NEGOTIATE_MESSAGE,CHALLENGE_MESSAGE,AUTHENTICATE_MESSAGE)
	1:	j:=0;
		FOR i:= 0 TO session^.NegMessByteLen - 1 DO
			temp[i] := session^.NegMessByte[j];
			j:=j+1;
		END_FOR
		j:=0;
		FOR i:= i TO session^.NegMessByteLen - 1 + session^.challMessByteLen DO
			temp[i] := session^.ChallMessByte[j];
			j:=j+1;
		END_FOR
		j:=0;
		FOR i:= i TO session^.NegMessByteLen - 1 + session^.challMessByteLen + session^.AuthMessByteLen DO
			temp[i] := session^.AuthMessByte[j];
			j:=j+1;
		END_FOR
		step:=2;

	2:	// Hash Concat with exported Session Key
		HMACMD5(key:=ADR(session^.exportedSessionKey),lenKey:=16,message:=ADR(temp),lenMess:=i,out=>out);
		HMACMD5.xExecute:= TRUE;
	
	IF HMACMD5.xDone THEN
		HMACMD5.xExecute:= TRUE;	
		xDone := TRUE;
		Step:=0;
	END_IF
	
END_CASE

END_FUNCTION_BLOCK

// Device/Application/Bausteine/SMB2_Client/NTLM/Functions/Hash/Encryption/HMAC_MD5
FUNCTION_BLOCK HMAC_MD5
VAR_INPUT
	xExecute:BOOL; // Start
	key:POINTER TO ARRAY[0..127] OF BYTE; // Key for Hash
	lenKey:INT; // Length of Key
	message:POINTER TO ARRAY[0..1024] OF BYTE; // Message for Hash
	lenMess:INT; // Length of Message
END_VAR
VAR_OUTPUT
	out:ARRAY[0..15] OF BYTE;
	xDone:BOOL;
END_VAR
VAR
	Step:INT;
	i:INT;
	keyX: ARRAY[0..63] OF BYTE;
	o_key_pad:ARRAY[0..63] OF BYTE;
	i_key_pad:ARRAY[0..63] OF BYTE;
	Temp:ARRAY[0..2048] OF BYTE;
	hashTemp:ARRAY[0..15] OF BYTE;
	hash: MEM.MD5;
END_VAR
VAR CONSTANT
	BLOCKSIZE:INT:= 64;
END_VAR

// Routine from Wikipedia  
// Keys longer than blocksize are shortened by hashing them
 //  if (length(key) > blocksize) then
  //    key ← hash(key) //Key becomes blocksize bytes long
   
 //  Keys shorter than blocksize are padded to blocksize by padding with zeros on the right
  // if (length(key) < blocksize) then
   //   key ← Pad(key, blocksize)  //pad key with zeros to make it blocksize bytes long
    
 //   o_key_pad = key xor [0x5c * blocksize]   //Outer padded key
 //   i_key_pad = key xor [0x36 * blocksize]   //Inner padded key
    
 //   return hash(o_key_pad ∥ hash(i_key_pad ∥ message)) //Where ∥ is concatenation


xDone:= FALSE;

CASE Step OF
0:	IF xExecute THEN
		Step:=1;
	END_IF

1:	 // Init key Array
	FOR i:=0 TO 63 DO
		keyX[i] := 0;
	END_FOR

	// key length match blocksize
	IF lenKey > BLOCKSIZE THEN
		RETURN;
	ELSIF lenKey < BLOCKSIZE THEN
		FOR i:=0 TO lenKey-1 DO
			keyX[i] := key^[i]; // Key + padding
		END_FOR
	END_IF
	
	FOR i:=0 TO BLOCKSIZE-1 DO
		o_key_pad[i] := keyX[i] XOR 16#5C; //Outer padded key
		i_key_pad[i] := keyX[i] XOR 16#36; //Inner padded key
	END_FOR
	
	Step:= 2;
	
2:	// Concat i_key_pad ∥ message
	FOR i:=0 TO BLOCKSIZE-1 DO
		Temp[i] := i_key_pad[i];
	END_FOR
	FOR i:=BLOCKSIZE TO BLOCKSIZE+lenMess DO
		Temp[i]:= message^[i-BLOCKSIZE];
	END_FOR
	
	step:= 3;
	
3:	// hash(i_key_pad ∥ message)
	hash(pMemoryBlock:=ADR(Temp[0]),udiNumberOfBytes:=INT_TO_UDINT(BLOCKSIZE+lenMess),abyDigest=>hashTemp);
	hash.xExecute:= TRUE;
	
	IF hash.xDone THEN
		step:= 4;
		hash.xExecute:= FALSE;
	END_IF
	
4:	// Conact o_key_pad and already hashed
	FOR i:=0 TO BLOCKSIZE-1 DO
		Temp[i] := o_key_pad[i];
	END_FOR
	FOR i:=BLOCKSIZE TO BLOCKSIZE+16 DO
		Temp[i]:= hashTemp[i-BLOCKSIZE];
	END_FOR
	
	Step:=5;
	
5:	// hash(o_key_pad ∥ hash(i_key_pad ∥ message))
	hash(pMemoryBlock:=ADR(Temp[0]),udiNumberOfBytes:=INT_TO_UDINT(BLOCKSIZE+16),abyDigest=>hashTemp);
	hash.xExecute:= TRUE;
	
	IF hash.xDone THEN
		step:= 0;
		hash.xExecute:= FALSE;
		FOR i:=0 TO 15 DO
			out[i] := hashTemp[i]; // Copy Hash to out variable
		END_FOR
		xDone:= TRUE;
	END_IF
END_CASE

END_FUNCTION_BLOCK

// Device/Application/Bausteine/SMB2_Client/NTLM/Functions/GetAVPairList
FUNCTION GetAVPairList : AVPairList
VAR_INPUT
	pSource:POINTER TO ARRAY[0..32767] OF BYTE; // Pointer to Start if Attribte List / Target Info
	ChallMess:POINTER TO CHALLENGE_MESSAGE; // Challenge Message
END_VAR

VAR
	i:INT;
	j:INT;
	len:INT;
	pLen:POINTER TO ARRAY[0..1] OF BYTE;
	pVar:POINTER TO ARRAY[0..32767] OF BYTE;
	Placeholder:WSTRING(80);
	terminateString:BOOL;
END_VAR
VAR CONSTANT
	MsvAvEOL:BYTE:=16#00;
	MsvAvNbComputerName:BYTE:=16#01;
	MsvAvNbDomainName:BYTE:=16#02;
	MsvAvDnsComputerName:BYTE:=16#03;
	MsvAvDnsDomainName:BYTE:=16#04;
	MsvAvDnsTreeName:BYTE:=16#05;
	MsvAvFlags:BYTE:=16#06;
	MsvAvTimestamp:BYTE:=16#07;
	MsvAvSingleHost:BYTE:=16#08;
	MsvAvTargetName:BYTE:=16#09;
	MsvChannelBindings:BYTE:=16#0A;
END_VAR

// This Function decodes the Attributes of Challene Message

pLen:= ADR(len); // length of Attribute List
pVar:=ADR(ChallMess^.AVPairListPayload[0]); 

FOR i:=0 TO WORD_TO_INT(ChallMess^.TargetInfoLen)-1 DO // Copy Source to ChallMess Struct
	pVar^[i] := pSource^[i];
END_FOR
	i:=0;
WHILE i <= WORD_TO_INT(ChallMess^.TargetInfoLen) DO 
	// Decode all Attributes
	CASE pSource^[i] OF   // Attribute Number?
	MsvAvEOL: EXIT;
	MsvAvNbComputerName: 	pVar:=ADR(ChallMess^.AVPairList.NBComputerName); terminateString:=TRUE;
	MsvAvNbDomainName:		pVar:=ADR(ChallMess^.AVPairList.NBDomainName);	terminateString:=TRUE;
	MsvAvDnsComputerName:	pVar:=ADR(ChallMess^.AVPairList.DNSComputerName); terminateString:=TRUE;
	MsvAvDnsDomainName:		pVar:=ADR(ChallMess^.AVPairList.DNSDomainName);	terminateString:=TRUE;
	MsvAvDnsTreeName:		pVar:=ADR(Placeholder);
	MsvAvFlags:				pVar:=ADR(Placeholder);
	MsvAvTimestamp:			pVar:=ADR(ChallMess^.AVPairList.TimeStamp[0]); GetAVPairList.xTimeStamp:= TRUE;
	MsvAvSingleHost:		pVar:=ADR(Placeholder);
	MsvAvTargetName:		pVar:=ADR(Placeholder);
	MsvChannelBindings:		pVar:=ADR(Placeholder);
	END_CASE
	
	// Decode Length and String
	i:=i+2;
	pLen^[0]:= pSource^[i]; pLen^[1]:= pSource^[i+1]; 
	i:= i+2;
	FOR j:=0 TO len-1 DO
		pVar^[j] := pSource^[i];
		i:= i+1;
		END_FOR
	// String Termination
	IF terminateString THEN
		pVar^[j]:= 0; pVar^[j+1]:= 0; 
		terminateString:=FALSE;
	END_IF
		
END_WHILE

END_FUNCTION

// Device/Application/Bausteine/SMB2_Client/NTLM/Functions/mechListMIC
FUNCTION_BLOCK mechListMIC
VAR_INPUT
	xExecute:BOOL; // Start
	session:POINTER TO SessionData; // NTLM Parameter
END_VAR
VAR_OUTPUT
	out:ARRAY[0..19] OF BYTE;
	xDone:BOOL;
END_VAR
VAR
	step:int:=0;
	temp:ARRAY[0..15] OF BYTE;
	RC4temp:ARRAY[0..15] OF BYTE;
	j:INT;
	i:INT;
	HMACMD5:HMAC_MD5;
	RC4K:RC4;
	MechTypeList:ARRAY[0..17] OF BYTE:= [16#00, 16#00, 16#00, 16#00, 16#30, 16#0C, 16#06, 16#0A, 16#2B, 16#06, 16#01, 16#04, 16#01, 16#82, 16#37, 16#02, 16#02, 16#0A]; // For this implementation only 1 MachType (NTLM)
	concat:ARRAY[0..7] OF BYTE:=[16#A3, 16#12, 16#04, 16#10, 16#01, 16#00, 16#00, 16#00];
END_VAR

// This Message generates the MechListMic from the MechList in Negotiate Message

xDone := FALSE;
IF Step = 0 AND xExecute = 1 THEN
	Step:=1;
END_IF
CASE step OF
	1:	j:=0;
		HMACMD5(key:=ADR(session^.ClientSigningKey),lenKey:=16,message:=ADR(MechTypeList),lenMess:=18,out=>temp); // Hash MechListMic mit Client Signing Key, MechListMic ist Static
		HMACMD5.xExecute:= TRUE;
		
		IF HMACMD5.xDone THEN
			HMACMD5.xExecute:= TRUE;	
			Step:=2;
		END_IF

	2:	RC4K(key:=ADR(session^.ClientSealingKey),lenKey:=16,data:=ADR(temp),lenData:=8,ciper:=ADR(RC4temp),Mode:=2); // RC4 over previous Hashed mit Client Sealing Key
		
		j:=0;
		// Concat Identifier with calculated
		FOR i:=0 TO 7 DO
			out[i] := concat[j];
			j:=j+1;
		END_FOR	
		j:=0;
		FOR i:=i TO 7+8 DO
			out[i] := RC4temp[j];
			j:=j+1;
		END_FOR	
		j:=0;
		FOR i:=i TO 7+8+4 DO
			out[i] := 0;
			j:=j+1;
		END_FOR	
	
		xDone:=TRUE;
		step:=0;
	
END_CASE

END_FUNCTION_BLOCK

// Device/Application/Bausteine/SMB2_Client/NTLM/Functions/Hash/Encryption/RC4
FUNCTION_BLOCK RC4
VAR_INPUT
	key:POINTER TO ARRAY[0..255] OF BYTE;
	lenKey:INT;
	data:POINTER TO ARRAY[0..32767] OF BYTE;
	lenData:INT;
	ciper:POINTER TO ARRAY[0..32767] OF BYTE;
	Mode:INT;
END_VAR
VAR_OUTPUT
END_VAR
VAR
	sbox:ARRAY[0..255] OF BYTE;
	i:INT;
	j:INT;
	n:INT;
	tempByte:BYTE;
	zufallszahl:BYTE;
END_VAR

// Mode 0, Init
IF mode = 0 OR mode=2 THEN
	FOR i:=0 TO 255 DO
		sbox[i] := INT_TO_BYTE(i);
	END_FOR
	j:=	0;
	
	FOR i:=0 TO 255 DO
		j:= (j + sbox[i] + key^[i MOD lenKey]) MOD 256;
		tempByte:= sbox[i];
		sbox[i] := sbox[j];
		sbox[j] := tempByte;
	END_FOR	
END_IF

// Mode 1, Streamcipher
IF mode = 1 OR mode=2 THEN
	i:= 0;
	j:= 0;
	
	FOR n:=0 TO lenData-1 DO
		i:= (i + 1) MOD 256;
		j:= (j + sbox[i]) MOD 256;
		tempByte:= sbox[i];
		sbox[i] := sbox[j];
		sbox[j] := tempByte;
		zufallszahl := sbox[(sbox[i]+sbox[j]) MOD 256];
		ciper^[n]:= zufallszahl XOR data^[n];
	END_FOR
END_IF

END_FUNCTION_BLOCK

// Device/Application/Bausteine/SMB2_Client/NTLM/Functions/GenerateAuthenticateMessage
FUNCTION_BLOCK GenerateAuthenticateMessage
VAR_INPUT
	session:POINTER TO sessionData; // NTLM Parameter
END_VAR
VAR_OUTPUT
	authMess:AUTHENTICATE_MESSAGE;
END_VAR
VAR
	i:INT;
	j:INT;
	sizePayload:INT;
	pVar:POINTER TO ARRAY[0..512] OF BYTE;
	pAuth:POINTER TO ARRAY[0..512] OF BYTE;
	tempLen:int;
END_VAR

// This Function generates the Auth Message and copied it to Struct

// Domain Name
	authMess.DomainNameLen:= INT_TO_WORD(wlen(session^.userDomain))*2;
	authMess.DomainNameMaxLen:=authMess.DomainNameLen;
	authMess.DomainNameBufferOffset:= 88;
	
// UserName
	authMess.UserNameLen:= INT_TO_WORD(wlen(session^.user))*2;
	authMess.UserNameMaxLen:=authMess.UserNameLen;
	authMess.UserNameBufferOffset:= authMess.DomainNameBufferOffset+authMess.DomainNameLen;
	
// Workstation
	authMess.WorkstationLen:= INT_TO_WORD(wlen(session^.userDomain))*2;
	authMess.WorkstationMaxLen:=authMess.WorkstationLen;
	authMess.WorkstationBufferOffset:= authMess.UserNameBufferOffset+authMess.UserNameLen;
	
// LmChallengeResponseFields
	authMess.LmChallengeResponseLen:= session^.lmChallengeResponseLen;
	authMess.LmChallengeResponseMaxLen:= session^.lmChallengeResponseLen;
	authMess.LmChallengeResponseBufferOffset:= authMess.WorkstationBufferOffset+authMess.WorkstationLen;
	
// NtChallengeResponseFields
	authMess.NtChallengeResponseLen:= session^.NtChallengeResponseLen;
	authMess.NtChallengeResponseMaxLen:= session^.NtChallengeResponseLen;
	authMess.NtChallengeResponseBufferOffset:= authMess.LmChallengeResponseBufferOffset+authMess.LmChallengeResponseLen;

// SessionKey
	authMess.EncryptedRandomSessionKeyLen:= 16;
	authMess.EncryptedRandomSessionKeyMaxLen:=16;
	authMess.EncryptedRandomSessionKeyBufferOffset:= authMess.NtChallengeResponseBufferOffset+authMess.NtChallengeResponseLen;

// NegotiateFlags 
	authMess.NegotiateFlags := session^.NegotiateFlags;
	
//	MIC, zero for MIC Calculation over whole Message
	FOR i:=0 TO 15 DO
		authMess.MIC[i]:= 0;
	END_FOR
	
	authMess.PayLoadSize:= UDINT_TO_INT (authMess.EncryptedRandomSessionKeyBufferOffset + authMess.EncryptedRandomSessionKeyLen); // Payload Size
	
	// Copy Data into Payloadbuffer
	j:=0;
	pVar:= ADR(session^.userDomain);
	FOR i:=0 TO WORD_TO_INT(authMess.DomainNameLen)-1 DO // Copy User Domain
		authMess.Payload[j] := pVar^[i];
		j:= j+1;
	END_FOR
	pVar:= ADR(session^.user);
	FOR i:=0 TO WORD_TO_INT(authMess.UserNameLen)-1 DO // Copy User
		authMess.Payload[j] := pVar^[i];
		j:= j+1;
	END_FOR
	pVar:= ADR(session^.userDomain);
	FOR i:=0 TO WORD_TO_INT(authMess.DomainNameLen)-1 DO // Copy User Domain
		authMess.Payload[j] := pVar^[i];
		j:= j+1;
	END_FOR
	pVar:= ADR(session^.lmChallengeResponse);
	FOR i:=0 TO WORD_TO_INT(authMess.LmChallengeResponseLen)-1 DO // Copy LM Challenge Response
		authMess.Payload[j] := pVar^[i];
		j:= j+1;
	END_FOR
	pVar:= ADR(session^.ntChallengeResponse);
	FOR i:=0 TO WORD_TO_INT(authMess.ntChallengeResponseLen)-1 DO // Copy NT Challenge Response
		authMess.Payload[j] := pVar^[i];
		j:= j+1;
	END_FOR
	pVar:= ADR(session^.encryptedRandomSessionKey);
	FOR i:=0 TO WORD_TO_INT(authMess.EncryptedRandomSessionKeyLen)-1 DO // Copy encrypted Random Session Key
		authMess.Payload[j] := pVar^[i];
		j:= j+1;
	END_FOR
	
	authMess.PayLoadSize := j;
	
	// Copy Auth Message into Struct
	pAuth:=ADR(AuthMess);
	tempLen:=88;
	FOR i:=0 TO tempLen-1 DO
		session^.AuthMessByte[i]:= pAuth^[i];
	END_FOR
		
	// Copy Auth Payload into struct
	pAuth:=ADR(AuthMess.Payload);
	tempLen:=88;
	FOR i:=0 TO AuthMess.PayLoadSize-1 DO
		session^.AuthMessByte[i+88]:= pAuth^[i];
	END_FOR
	
	session^.AuthMessByteLen := 88+AuthMess.PayLoadSize; // Length of Auth Message

END_FUNCTION_BLOCK

// Device/Application/Bausteine/SMB2_Client/Misc/DER_Encoding
FUNCTION_BLOCK DER_Encoding
VAR_INPUT
	pDest:POINTER TO BYTE;
	Length:INT;
	TestLen:BOOL;
END_VAR
VAR_OUTPUT
	pOut:POINTER TO BYTE;
	NumOct:INT;
END_VAR
VAR
	tempByte:byte;
	pVar: POINTER TO BYTE;
END_VAR


pVar:=pDest;
IF TestLen= FALSE THEN
	IF Length < 128 THEN
		pVar^:=UINT_TO_BYTE(INT_TO_UINT(Length) AND 16#007F);
		pOut:= pVar+1;
	ELSIF Length >= 128 AND Length <= 255 THEN
		pVar^:= 16#81; // 1 Octets
		pVar:=pVar + 1;
		pVar^:= UINT_TO_BYTE(INT_TO_UINT(Length) AND 16#00FF);
		pOut:= pVar+1;
	ELSIF Length > 255 AND Length <= 65535 THEN
		pVar^:= 16#82; // 2 Octets
		pVar:=pVar + 1;
		pVar^:= UINT_TO_BYTE(SHR(INT_TO_UINT(Length),8) AND 16#00FF);
		pVar:=pVar + 1;
		pVar^:= UINT_TO_BYTE(INT_TO_UINT(Length) AND 16#00FF);
		pOut:= pVar+1;
	END_IF
ELSIF TestLen= TRUE THEN
	IF Length < 128 THEN
	NumOct:= 1+1;
	ELSIF Length >= 128 AND Length <= 255 THEN
	NumOct:= 2+1;
	ELSIF Length > 255 AND Length <= 65535 THEN
	NumOct:= 3+1;
	END_IF
END_IF

END_FUNCTION_BLOCK

// Device/Application/Bausteine/SMB2_Client/Misc/DER_Len
FUNCTION_BLOCK DER_Len
VAR_INPUT
	pSource:POINTER TO BYTE;
END_VAR
VAR_OUTPUT
	pOut:POINTER TO BYTE;
	Length:INT;
END_VAR
VAR
	pVar: POINTER TO BYTE;
	tempINT:INT;
	NumberOct:INT;
END_VAR


pVar:=pSource;

IF pVar^ < 128 THEN // TokenLength
	tempINT := pVar^;
	Length := UINT_TO_INT(INT_TO_UINT(tempINT) AND 16#7F);
	pVar := pVar+1;
ELSE			
	NumberOct:= pVar^ AND 16#7F;
	pVar := pVar+1;
END_IF

//pVar:= pVar+1;

// Decode Length
IF NumberOct = 1 THEN // 1 Octet
	Length := pVar^;
ELSIF NumberOct = 2 THEN // 2 Octet
	tempINT := UINT_TO_INT(SHL(BYTE_TO_UINT(pVar^),8) AND 16#FF00);
	pVar:= pVar+1;
	Length := tempINT + UINT_TO_INT((BYTE_TO_UINT(pVar^) AND 16#FF));
END_IF

pOut:= pVar+1;

END_FUNCTION_BLOCK

